  MoveC 664 to (45.79, 82.06, -1) mm, rotated rx -180 ry 0 rz 90 deg; joints [76.857, -17.355, 82.878, 0, 24.477, 76.857] to (20.03, 82.47, -1) mm, rotated rx -180 ry 0 rz 90 deg; joints [76.673, -17.853, 84.752, 0, 23.101, 76.673]
  MoveL 665 to (19.93, 74.92, -1) mm, rotated rx 180 ry 0 rz 90 deg; joints [76.425, -17.821, 84.63, 0, 23.192, 76.425]
  MoveL 666 to (19.93, 74.92, 2) mm, rotated rx 180 ry 0 rz 90 deg; joints [76.425, -17.975, 84.73, 0, 23.244, 76.425]
  Establecer velocidad (1000.0 mm/s)
  MoveL 667 to (19.93, 74.92, 10) mm, rotated rx 180 ry 0 rz 90 deg; joints [76.425, -18.384, 84.996, 0, 23.387, 76.425]
  Establecer velocidad (66.7 mm/s)
  MoveL 668 to (26.55, 73.47, 10) mm, rotated rx -180 ry 0 rz 90 deg; joints [76.43, -18.251, 84.495, 0, 23.756, 76.43]
  MoveL 669 to (26.55, 73.47, 2) mm, rotated rx 180 ry 0 rz 90 deg; joints [76.43, -17.843, 84.229, 0, 23.614, 76.43]
  MoveL 670 to (26.75, 74.97, 1.59) mm, rotated rx -180 ry 0 rz 90 deg; joints [76.48, -17.825, 84.227, 0, 23.598, 76.48]
  MoveL 671 to (26.59, 76.48, 1.19) mm, rotated rx -180 ry 0 rz 90 deg; joints [76.529, -17.815, 84.251, 0, 23.563, 76.529]
  MoveL 672 to (26.1, 77.92, 0.78) mm, rotated rx 180 ry 0 rz 90 deg; joints [76.572, -17.81, 84.298, 0, 23.512, 76.572]
  MoveL 673 to (25.3, 79.21, 0.38) mm, rotated rx 180 ry 0 rz 90 deg; joints [76.608, -17.81, 84.364, 0, 23.446, 76.608]
  MoveL 674 to (24.24, 80.3, -0.03) mm, rotated rx -180 ry 0 rz 90 deg; joints [76.635, -17.814, 84.446, 0, 23.369, 76.635]
  MoveL 675 to (22.96, 81.12, -0.44) mm, rotated rx 180 ry 0 rz 90 deg; joints [76.652, -17.821, 84.538, 0, 23.283, 76.652]
  MoveL 676 to (21.53, 81.64, -0.84) mm, rotated rx 180 ry 0 rz 90 deg; joints [76.658, -17.83, 84.636, 0, 23.194, 76.658]
  MoveL 677 to (20.02, 81.8, -1.25) mm, rotated rx 180 ry 0 rz 90 deg; joints [76.651, -17.838, 84.733, 0, 23.105, 76.651]
  MoveC 678 to (-5.39, 82.11, -1.25) mm, rotated rx 180 ry 0 rz 90 deg; joints [76.461, -18.297, 86.542, 0, 21.755, 76.461] to (-30.8, 82.31, -1.25) mm, rotated rx 180 ry 0 rz 90 deg; joints [76.261, -18.726, 88.313, 0, 20.412, 76.261]
  MoveC 679 to (-35.67, 81.83, -1.25) mm, rotated rx 180 ry 0 rz 90 deg; joints [76.205, -18.803, 88.641, 0, 20.162, 76.205] to (-40.33, 80.31, -1.25) mm, rotated rx -180 ry 0 rz 90 deg; joints [76.115, -18.871, 88.934, 0, 19.937, 76.115]
  MoveC 680 to (-44.55, 75.38, -1.25) mm, rotated rx 180 ry 0 rz 90 deg; joints [75.912, -18.918, 89.138, 0, 19.779, 75.912] to (-43.44, 68.99, -1.25) mm, rotated rx -180 ry 0 rz 90 deg; joints [75.705, -18.875, 88.953, 0, 19.922, 75.705]
  MoveC 681 to (-40.9, 66.02, -1.25) mm, rotated rx 180 ry 0 rz 90 deg; joints [75.627, -18.823, 88.727, 0, 20.096, 75.627] to (-37.82, 63.61, -1.25) mm, rotated rx 180 ry 0 rz 90 deg; joints [75.572, -18.763, 88.473, 0, 20.29, 75.572]
  MoveL 682 to (-14.69, 48.96, -1.25) mm, rotated rx 180 ry 0 rz 90 deg; joints [75.284, -18.314, 86.609, 0, 21.705, 75.284]
  MoveC 683 to (-10.76, 47.27, -1.25) mm, rotated rx -180 ry 0 rz 90 deg; joints [75.262, -18.238, 86.303, 0, 21.935, 75.262] to (-6.49, 46.9, -1.25) mm, rotated rx 180 ry 0 rz 90 deg; joints [75.287, -18.161, 85.996, 0, 22.165, 75.287]
  MoveL 684 to (63.97, 51.98, -1.25) mm, rotated rx 180 ry 0 rz 90 deg; joints [76.033, -16.822, 80.991, 0, 25.832, 76.033]
  MoveL 685 to (72.21, 52.56, -1.25) mm, rotated rx 180 ry 0 rz 90 deg; joints [76.117, -16.65, 80.385, 0, 26.266, 76.117]
  MoveC 686 to (77.75, 55.2, -1.25) mm, rotated rx 180 ry 0 rz 90 deg; joints [76.243, -16.545, 80.016, 0, 26.528, 76.243] to (80, 60.92, -1.25) mm, rotated rx -180 ry 0 rz 90 deg; joints [76.441, -16.526, 79.951, 0, 26.575, 76.441]
  MoveL 687 to (80, 72.47, -1.25) mm, rotated rx -180 ry 0 rz 90 deg; joints [76.806, -16.586, 80.159, 0, 26.426, 76.806]
  MoveC 688 to (77.62, 78.32, -1.25) mm, rotated rx -180 ry 0 rz 90 deg; joints [76.974, -16.667, 80.442, 0, 26.225, 76.974] to (71.82, 80.84, -1.25) mm, rotated rx -180 ry 0 rz 90 deg; joints [77.012, -16.803, 80.92, 0, 25.882, 77.012]
  MoveC 689 to (45.92, 81.38, -1.25) mm, rotated rx 180 ry 0 rz 90 deg; joints [76.836, -17.337, 82.848, 0, 24.488, 76.836] to (20.02, 81.8, -1.25) mm, rotated rx 180 ry 0 rz 90 deg; joints [76.651, -17.838, 84.733, 0, 23.105, 76.651]
  MoveL 690 to (19.92, 74.25, -1.25) mm, rotated rx 180 ry 0 rz 90 deg; joints [76.403, -17.806, 84.611, 0, 23.195, 76.403]
  MoveL 691 to (19.92, 74.25, 1.75) mm, rotated rx 180 ry 0 rz 90 deg; joints [76.403, -17.959, 84.711, 0, 23.248, 76.403]
  Establecer velocidad (1000.0 mm/s)
  MoveL 692 to (19.92, 74.25, 10) mm, rotated rx 180 ry 0 rz 90 deg; joints [76.403, -18.381, 84.985, 0, 23.395, 76.403]
  Establecer velocidad (66.7 mm/s)
  MoveL 693 to (38.36, 29.5, 10) mm, rotated rx -180 ry 0 rz 90 deg; joints [75.107, -17.799, 82.829, 0, 24.97, 75.107]
  MoveL 694 to (38.36, 29.5, 2) mm, rotated rx -180 ry 0 rz 90 deg; joints [75.107, -17.394, 82.562, 0, 24.831, 75.107]
  MoveL 695 to (38.51, 31.01, 1.59) mm, rotated rx -180 ry 0 rz 90 deg; joints [75.156, -17.378, 82.567, 0, 24.811, 75.156]
  MoveL 696 to (38.29, 32.51, 1.19) mm, rotated rx -180 ry 0 rz 90 deg; joints [75.203, -17.37, 82.599, 0, 24.771, 75.203]
  MoveL 697 to (37.74, 33.93, 0.78) mm, rotated rx 180 ry 0 rz 90 deg; joints [75.243, -17.368, 82.653, 0, 24.715, 75.243]
  MoveL 698 to (36.89, 35.19, 0.38) mm, rotated rx 180 ry 0 rz 90 deg; joints [75.277, -17.371, 82.725, 0, 24.646, 75.277]
  MoveL 699 to (35.78, 36.23, -0.03) mm, rotated rx -180 ry 0 rz 90 deg; joints [75.301, -17.378, 82.812, 0, 24.566, 75.301]
  MoveL 700 to (34.47, 37, -0.44) mm, rotated rx -180 ry 0 rz 90 deg; joints [75.314, -17.387, 82.909, 0, 24.478, 75.314]
  MoveL 701 to (33.02, 37.46, -0.84) mm, rotated rx 180 ry 0 rz 90 deg; joints [75.317, -17.397, 83.009, 0, 24.388, 75.317]
  MoveL 702 to (31.51, 37.56, -1.25) mm, rotated rx -180 ry 0 rz 90 deg; joints [75.307, -17.407, 83.107, 0, 24.3, 75.307]
  MoveL 703 to (7.58, 36.92, -1.25) mm, rotated rx 180 ry 0 rz 90 deg; joints [75.082, -17.859, 84.815, 0, 23.044, 75.082]
  MoveC 704 to (3.41, 36.01, -1.25) mm, rotated rx 180 ry 0 rz 90 deg; joints [75.016, -17.931, 85.093, 0, 22.838, 75.016] to (-0.13, 33.64, -1.25) mm, rotated rx -180 ry 0 rz 90 deg; joints [74.908, -17.984, 85.299, 0, 22.685, 74.908]
  MoveC 705 to (-2.38, 29.17, -1.25) mm, rotated rx -180 ry 0 rz 90 deg; joints [74.741, -18.003, 85.373, 0, 22.63, 74.741] to (-2.11, 24.17, -1.25) mm, rotated rx 180 ry 0 rz 90 deg; joints [74.581, -17.973, 85.256, 0, 22.717, 74.581]
  MoveL 706 to (-1.81, 23.22, -1.25) mm, rotated rx 180 ry 0 rz 90 deg; joints [74.552, -17.963, 85.217, 0, 22.746, 74.552]
  MoveL 707 to (3.68, 8.05, -1.25) mm, rotated rx 180 ry 0 rz 90 deg; joints [74.11, -17.784, 84.526, 0, 23.257, 74.11]
  MoveL 708 to (4.33, 6.33, -1.25) mm, rotated rx 180 ry 0 rz 90 deg; joints [74.06, -17.763, 84.446, 0, 23.317, 74.06]
  MoveC 709 to (5.69, 3.82, -1.25) mm, rotated rx -180 ry 0 rz 90 deg; joints [73.992, -17.724, 84.297, 0, 23.427, 73.992] to (7.69, 1.78, -1.25) mm, rotated rx -180 ry 0 rz 90 deg; joints [73.944, -17.675, 84.113, 0, 23.562, 73.944]
  MoveL 710 to (25.11, -11.75, -1.25) mm, rotated rx 180 ry 0 rz 90 deg; joints [73.673, -17.263, 82.579, 0, 24.685, 73.673]
  MoveC 711 to (32.35, -13.71, -1.25) mm, rotated rx -180 ry 0 rz 90 deg; joints [73.678, -17.107, 82.011, 0, 25.096, 73.678] to (38.84, -9.95, -1.25) mm, rotated rx 180 ry 0 rz 90 deg; joints [73.857, -16.998, 81.617, 0, 25.381, 73.857]
  MoveL 712 to (39.33, -9.33, -1.25) mm, rotated rx 180 ry 0 rz 90 deg; joints [73.881, -16.992, 81.594, 0, 25.397, 73.881]
  MoveL 713 to (62.07, 22.39, -1.25) mm, rotated rx 180 ry 0 rz 90 deg; joints [75.082, -16.701, 80.564, 0, 26.137, 75.082]
  MoveL 714 to (62.82, 23.49, -1.25) mm, rotated rx 180 ry 0 rz 90 deg; joints [75.123, -16.692, 80.53, 0, 26.162, 75.123]
  MoveC 715 to (64.55, 27.94, -1.25) mm, rotated rx 180 ry 0 rz 90 deg; joints [75.277, -16.68, 80.488, 0, 26.191, 75.277] to (64.19, 32.69, -1.25) mm, rotated rx 180 ry 0 rz 90 deg; joints [75.424, -16.714, 80.608, 0, 26.106, 75.424]
  MoveC 716 to (60.61, 36.69, -1.25) mm, rotated rx 180 ry 0 rz 90 deg; joints [75.521, -16.812, 80.952, 0, 25.859, 75.521] to (55.44, 38.13, -1.25) mm, rotated rx 180 ry 0 rz 90 deg; joints [75.525, -16.927, 81.364, 0, 25.564, 75.525]
  MoveL 717 to (53.54, 38.15, -1.25) mm, rotated rx -180 ry 0 rz 90 deg; joints [75.51, -16.967, 81.504, 0, 25.462, 75.51]
  MoveL 718 to (31.51, 37.56, -1.25) mm, rotated rx -180 ry 0 rz 90 deg; joints [75.307, -17.407, 83.107, 0, 24.3, 75.307]
  MoveL 719 to (31.71, 30.01, -1.25) mm, rotated rx -180 ry 0 rz 90 deg; joints [75.066, -17.364, 82.948, 0, 24.416, 75.066]
  MoveL 720 to (31.71, 30.01, 1.75) mm, rotated rx 180 ry 0 rz 90 deg; joints [75.066, -17.516, 83.048, 0, 24.468, 75.066]
  Establecer velocidad (1000.0 mm/s)
  MoveL 721 to (31.71, 30.01, 10) mm, rotated rx 180 ry 0 rz 90 deg; joints [75.066, -17.935, 83.323, 0, 24.612, 75.066]
  Establecer velocidad (66.7 mm/s)
  MoveL 722 to (72.21, -30.7, 10) mm, rotated rx 180 ry 0 rz 90 deg; joints [73.514, -16.719, 79.06, 0, 27.659, 73.514]
  MoveL 723 to (72.21, -30.7, 2) mm, rotated rx 180 ry 0 rz 90 deg; joints [73.514, -16.319, 78.791, 0, 27.527, 73.514]
  MoveL 724 to (73.71, -30.89, 1.59) mm, rotated rx 180 ry 0 rz 90 deg; joints [73.522, -16.263, 78.66, 0, 27.604, 73.522]
  MoveL 725 to (75.22, -30.71, 1.19) mm, rotated rx 180 ry 0 rz 90 deg; joints [73.541, -16.211, 78.536, 0, 27.675, 73.541]
  MoveL 726 to (76.65, -30.2, 0.78) mm, rotated rx 180 ry 0 rz 90 deg; joints [73.57, -16.161, 78.425, 0, 27.737, 73.57]
  MoveL 727 to (77.93, -29.38, 0.38) mm, rotated rx 180 ry 0 rz 90 deg; joints [73.607, -16.118, 78.332, 0, 27.786, 73.607]
  MoveL 728 to (79, -28.3, -0.03) mm, rotated rx -180 ry 0 rz 90 deg; joints [73.65, -16.08, 78.261, 0, 27.819, 73.65]
  MoveL 729 to (79.81, -27.01, -0.44) mm, rotated rx 180 ry 0 rz 90 deg; joints [73.697, -16.05, 78.215, 0, 27.836, 73.697]
  MoveL 730 to (80.31, -25.58, -0.84) mm, rotated rx 180 ry 0 rz 90 deg; joints [73.745, -16.028, 78.195, 0, 27.834, 73.745]
  MoveL 731 to (80.45, -24.06, -1.25) mm, rotated rx -180 ry 0 rz 90 deg; joints [73.793, -16.015, 78.204, 0, 27.811, 73.793]
  MoveL 732 to (80.45, -5.21, -1.25) mm, rotated rx 180 ry 0 rz 90 deg; joints [74.376, -16.136, 78.613, 0, 27.523, 74.376]
  MoveL 733 to (80.42, -3.53, -1.25) mm, rotated rx -180 ry 0 rz 90 deg; joints [74.427, -16.147, 78.651, 0, 27.496, 74.427]
  MoveC 734 to (80.02, -0.05, -1.25) mm, rotated rx 180 ry 0 rz 90 deg; joints [74.532, -16.178, 78.755, 0, 27.423, 74.532] to (78.95, 3.29, -1.25) mm, rotated rx 180 ry 0 rz 90 deg; joints [74.627, -16.222, 78.905, 0, 27.317, 74.627]
  MoveC 735 to (74.11, 7.51, -1.25) mm, rotated rx -180 ry 0 rz 90 deg; joints [74.717, -16.355, 79.359, 0, 26.995, 74.717] to (67.8, 6.36, -1.25) mm, rotated rx 180 ry 0 rz 90 deg; joints [74.627, -16.486, 79.811, 0, 26.675, 74.627]
  MoveC 736 to (65.35, 4.27, -1.25) mm, rotated rx 180 ry 0 rz 90 deg; joints [74.54, -16.526, 79.951, 0, 26.575, 74.54] to (63.25, 1.83, -1.25) mm, rotated rx -180 ry 0 rz 90 deg; joints [74.445, -16.557, 80.057, 0, 26.499, 74.445]
  MoveL 737 to (46.96, -20.52, -1.25) mm, rotated rx 180 ry 0 rz 90 deg; joints [73.599, -16.766, 80.793, 0, 25.974, 73.599]
  MoveC 738 to (45.17, -26.46, -1.25) mm, rotated rx 180 ry 0 rz 90 deg; joints [73.396, -16.767, 80.795, 0, 25.972, 73.396] to (47.5, -32.22, -1.25) mm, rotated rx -180 ry 0 rz 90 deg; joints [73.238, -16.682, 80.496, 0, 26.186, 73.238]
  MoveL 739 to (49.58, -34.59, -1.25) mm, rotated rx 180 ry 0 rz 90 deg; joints [73.183, -16.623, 80.288, 0, 26.334, 73.183]
  MoveL 740 to (62.07, -48.7, -1.25) mm, rotated rx 180 ry 0 rz 90 deg; joints [72.864, -16.26, 79.035, 0, 27.225, 72.864]
  MoveL 741 to (64.05, -50.95, -1.25) mm, rotated rx 180 ry 0 rz 90 deg; joints [72.814, -16.201, 78.834, 0, 27.367, 72.814]
  MoveC 742 to (66.41, -53.1, -1.25) mm, rotated rx -180 ry 0 rz 90 deg; joints [72.77, -16.134, 78.607, 0, 27.527, 72.77] to (69.17, -54.7, -1.25) mm, rotated rx -180 ry 0 rz 90 deg; joints [72.747, -16.061, 78.36, 0, 27.701, 72.747]
  MoveC 743 to (74.84, -54.84, -1.25) mm, rotated rx 180 ry 0 rz 90 deg; joints [72.797, -15.932, 77.928, 0, 28.005, 72.797] to (78.95, -50.94, -1.25) mm, rotated rx 180 ry 0 rz 90 deg; joints [72.955, -15.866, 77.706, 0, 28.16, 72.955]
  MoveC 744 to (79.99, -47.84, -1.25) mm, rotated rx 180 ry 0 rz 90 deg; joints [73.059, -15.864, 77.699, 0, 28.165, 73.059] to (80.41, -44.6, -1.25) mm, rotated rx 180 ry 0 rz 90 deg; joints [73.162, -15.877, 77.743, 0, 28.134, 73.162]
  MoveL 745 to (80.45, -43.12, -1.25) mm, rotated rx 180 ry 0 rz 90 deg; joints [73.208, -15.886, 77.773, 0, 28.113, 73.208]
  MoveL 746 to (80.45, -24.06, -1.25) mm, rotated rx -180 ry 0 rz 90 deg; joints [73.793, -16.015, 78.204, 0, 27.811, 73.793]
  MoveL 747 to (72.9, -24.06, -1.25) mm, rotated rx 180 ry 0 rz 90 deg; joints [73.725, -16.184, 78.777, 0, 27.407, 73.725]
  MoveL 748 to (72.9, -24.06, 1.75) mm, rotated rx -180 ry 0 rz 90 deg; joints [73.725, -16.334, 78.878, 0, 27.456, 73.725]
  Establecer velocidad (1000.0 mm/s)
  MoveL 749 to (72.9, -24.06, 10) mm, rotated rx 180 ry 0 rz 90 deg; joints [73.725, -16.747, 79.155, 0, 27.592, 73.725]
  Establecer velocidad (66.7 mm/s)
  MoveL 750 to (18.32, -73.74, 10) mm, rotated rx 180 ry 0 rz 90 deg; joints [71.653, -17.581, 82.045, 0, 25.536, 71.653]
  MoveL 751 to (18.32, -73.74, 2) mm, rotated rx 180 ry 0 rz 90 deg; joints [71.653, -17.177, 81.779, 0, 25.398, 71.653]
  MoveL 752 to (18.15, -75.25, 1.59) mm, rotated rx -180 ry 0 rz 90 deg; joints [71.604, -17.15, 81.741, 0, 25.409, 71.604]
  MoveL 753 to (18.35, -76.76, 1.19) mm, rotated rx -180 ry 0 rz 90 deg; joints [71.559, -17.115, 81.677, 0, 25.438, 71.559]
  MoveL 754 to (18.87, -78.18, 0.78) mm, rotated rx 180 ry 0 rz 90 deg; joints [71.52, -17.074, 81.591, 0, 25.484, 71.52]
  MoveL 755 to (19.7, -79.46, 0.38) mm, rotated rx 180 ry 0 rz 90 deg; joints [71.489, -17.028, 81.486, 0, 25.542, 71.489]
  MoveL 756 to (20.79, -80.51, -0.03) mm, rotated rx -180 ry 0 rz 90 deg; joints [71.467, -16.978, 81.368, 0, 25.611, 71.467]
  MoveL 757 to (22.09, -81.31, -0.44) mm, rotated rx -180 ry 0 rz 90 deg; joints [71.456, -16.926, 81.24, 0, 25.686, 71.456]
  MoveL 758 to (23.53, -81.79, -0.84) mm, rotated rx -180 ry 0 rz 90 deg; joints [71.456, -16.873, 81.11, 0, 25.762, 71.456]
  MoveL 759 to (25.04, -81.91, -1.25) mm, rotated rx 180 ry 0 rz 90 deg; joints [71.468, -16.82, 80.984, 0, 25.837, 71.468]
  MoveL 760 to (53.54, -81.62, -1.25) mm, rotated rx -180 ry 0 rz 90 deg; joints [71.769, -16.217, 78.888, 0, 27.329, 71.769]
  MoveL 761 to (55.06, -81.52, -1.25) mm, rotated rx 180 ry 0 rz 90 deg; joints [71.787, -16.184, 78.777, 0, 27.407, 71.787]
  MoveC 762 to (59.46, -80.25, -1.25) mm, rotated rx 180 ry 0 rz 90 deg; joints [71.87, -16.096, 78.478, 0, 27.618, 71.87] to (62.9, -77.23, -1.25) mm, rotated rx -180 ry 0 rz 90 deg; joints [71.997, -16.041, 78.294, 0, 27.748, 71.997]
  MoveC 763 to (63.97, -72.6, -1.25) mm, rotated rx 180 ry 0 rz 90 deg; joints [72.149, -16.051, 78.326, 0, 27.725, 72.149] to (62.62, -68.03, -1.25) mm, rotated rx -180 ry 0 rz 90 deg; joints [72.275, -16.114, 78.538, 0, 27.576, 72.275]
  MoveC 764 to (61.36, -66.14, -1.25) mm, rotated rx 180 ry 0 rz 90 deg; joints [72.321, -16.155, 78.678, 0, 27.477, 72.321] to (59.94, -64.36, -1.25) mm, rotated rx 180 ry 0 rz 90 deg; joints [72.362, -16.199, 78.827, 0, 27.372, 72.362]
  MoveL 765 to (32.58, -32.69, -1.25) mm, rotated rx 180 ry 0 rz 90 deg; joints [73.081, -16.988, 81.581, 0, 25.407, 73.081]
  MoveL 766 to (30.88, -30.8, -1.25) mm, rotated rx -180 ry 0 rz 90 deg; joints [73.125, -17.034, 81.747, 0, 25.287, 73.125]
  MoveL 767 to (30.8, -30.72, -1.25) mm, rotated rx 180 ry 0 rz 90 deg; joints [73.127, -17.036, 81.755, 0, 25.281, 73.127]
  MoveL 768 to (15.64, -18.58, -1.25) mm, rotated rx 180 ry 0 rz 90 deg; joints [73.367, -17.409, 83.117, 0, 24.293, 73.367]
  MoveL 769 to (14.69, -17.89, -1.25) mm, rotated rx -180 ry 0 rz 90 deg; joints [73.379, -17.432, 83.2, 0, 24.232, 73.379]
  MoveC 770 to (10.61, -16.09, -1.25) mm, rotated rx -180 ry 0 rz 90 deg; joints [73.398, -17.521, 83.53, 0, 23.99, 73.398] to (6.16, -16.06, -1.25) mm, rotated rx 180 ry 0 rz 90 deg; joints [73.356, -17.605, 83.849, 0, 23.757, 73.356]
  MoveC 771 to (1.83, -18.59, -1.25) mm, rotated rx 180 ry 0 rz 90 deg; joints [73.234, -17.673, 84.103, 0, 23.569, 73.234] to (-0.74, -22.9, -1.25) mm, rotated rx 180 ry 0 rz 90 deg; joints [73.07, -17.697, 84.193, 0, 23.503, 73.07]
  MoveL 772 to (-1.12, -24.17, -1.25) mm, rotated rx -180 ry 0 rz 90 deg; joints [73.026, -17.696, 84.192, 0, 23.504, 73.026]
  MoveL 773 to (-12.95, -68.7, -1.25) mm, rotated rx 180 ry 0 rz 90 deg; joints [71.483, -17.651, 84.021, 0, 23.63, 71.483]
  MoveL 774 to (-13.18, -69.65, -1.25) mm, rotated rx 180 ry 0 rz 90 deg; joints [71.45, -17.649, 84.015, 0, 23.635, 71.45]
  MoveC 775 to (-11.86, -77.67, -1.25) mm, rotated rx 180 ry 0 rz 90 deg; joints [71.21, -17.574, 83.731, 0, 23.843, 71.21] to (-4.97, -81.97, -1.25) mm, rotated rx -180 ry 0 rz 90 deg; joints [71.149, -17.416, 83.14, 0, 24.276, 71.149]
  MoveC 776 to (-3.18, -82.14, -1.25) mm, rotated rx 180 ry 0 rz 90 deg; joints [71.163, -17.38, 83.008, 0, 24.372, 71.163] to (-1.37, -82.19, -1.25) mm, rotated rx 180 ry 0 rz 90 deg; joints [71.181, -17.345, 82.879, 0, 24.466, 71.181]
  MoveL 777 to (25.04, -81.91, -1.25) mm, rotated rx 180 ry 0 rz 90 deg; joints [71.468, -16.82, 80.984, 0, 25.837, 71.468]
  MoveL 778 to (24.96, -74.36, -1.25) mm, rotated rx 180 ry 0 rz 90 deg; joints [71.702, -16.874, 81.172, 0, 25.701, 71.702]
  MoveL 779 to (24.96, -74.36, 1.75) mm, rotated rx -180 ry 0 rz 90 deg; joints [71.702, -17.025, 81.273, 0, 25.752, 71.702]
  Establecer velocidad (1000.0 mm/s)
  MoveL 780 to (24.96, -74.36, 10) mm, rotated rx -180 ry 0 rz 90 deg; joints [71.702, -17.441, 81.549, 0, 25.892, 71.702]
  Establecer velocidad (66.7 mm/s)
  MoveL 781 to (-60.08, -73.94, 10) mm, rotated rx -180 ry 0 rz 90 deg; joints [70.798, -19.029, 87.529, 0, 21.5, 70.798]
  MoveL 782 to (-60.08, -73.94, 2) mm, rotated rx 180 ry 0 rz 90 deg; joints [70.798, -18.616, 87.263, 0, 21.353, 70.798]
  MoveL 783 to (-60.25, -75.45, 1.59) mm, rotated rx -180 ry 0 rz 90 deg; joints [70.747, -18.589, 87.226, 0, 21.363, 70.747]
  MoveL 784 to (-60.06, -76.96, 1.19) mm, rotated rx 180 ry 0 rz 90 deg; joints [70.7, -18.556, 87.163, 0, 21.393, 70.7]
  MoveL 785 to (-59.53, -78.38, 0.78) mm, rotated rx 180 ry 0 rz 90 deg; joints [70.66, -18.518, 87.08, 0, 21.438, 70.66]
  MoveL 786 to (-58.7, -79.66, 0.38) mm, rotated rx -180 ry 0 rz 90 deg; joints [70.628, -18.476, 86.98, 0, 21.496, 70.628]
  MoveL 787 to (-57.62, -80.72, -0.03) mm, rotated rx -180 ry 0 rz 90 deg; joints [70.606, -18.43, 86.867, 0, 21.563, 70.606]
  MoveL 788 to (-56.32, -81.51, -0.44) mm, rotated rx -180 ry 0 rz 90 deg; joints [70.596, -18.383, 86.746, 0, 21.637, 70.596]
  MoveL 789 to (-54.88, -82, -0.84) mm, rotated rx 180 ry 0 rz 90 deg; joints [70.596, -18.335, 86.623, 0, 21.712, 70.596]
  MoveL 790 to (-53.37, -82.13, -1.25) mm, rotated rx 180 ry 0 rz 90 deg; joints [70.609, -18.288, 86.503, 0, 21.784, 70.609]
  MoveL 791 to (-36.48, -81.98, -1.25) mm, rotated rx 180 ry 0 rz 90 deg; joints [70.804, -17.996, 85.347, 0, 22.649, 70.804]
  MoveL 792 to (-35.19, -81.96, -1.25) mm, rotated rx -180 ry 0 rz 90 deg; joints [70.819, -17.973, 85.258, 0, 22.715, 70.819]
  MoveC 793 to (-28.29, -79.52, -1.25) mm, rotated rx 180 ry 0 rz 90 deg; joints [70.973, -17.865, 84.838, 0, 23.027, 70.973] to (-24.28, -73.41, -1.25) mm, rotated rx -180 ry 0 rz 90 deg; joints [71.212, -17.83, 84.705, 0, 23.126, 71.212]
  MoveL 794 to (-11.95, -26.06, -1.25) mm, rotated rx 180 ry 0 rz 90 deg; joints [72.858, -17.885, 84.916, 0, 22.969, 72.858]
  MoveL 795 to (-11.48, -24.17, -1.25) mm, rotated rx 180 ry 0 rz 90 deg; joints [72.924, -17.887, 84.924, 0, 22.963, 72.924]
  MoveC 796 to (-11.52, -18.64, -1.25) mm, rotated rx 180 ry 0 rz 90 deg; joints [73.102, -17.919, 85.045, 0, 22.873, 73.102] to (-14.07, -13.74, -1.25) mm, rotated rx 180 ry 0 rz 90 deg; joints [73.236, -17.991, 85.329, 0, 22.663, 73.236]
  MoveC 797 to (-18.74, -10.95, -1.25) mm, rotated rx 180 ry 0 rz 90 deg; joints [73.281, -18.09, 85.714, 0, 22.376, 73.281] to (-24.17, -10.71, -1.25) mm, rotated rx 180 ry 0 rz 90 deg; joints [73.235, -18.186, 86.097, 0, 22.089, 73.235]
  MoveL 798 to (-73.89, -21.27, -1.25) mm, rotated rx 180 ry 0 rz 90 deg; joints [72.38, -18.947, 89.266, 0, 19.681, 72.38]
  MoveC 799 to (-80.35, -25.23, -1.25) mm, rotated rx -180 ry 0 rz 90 deg; joints [72.179, -19.026, 89.613, 0, 19.413, 72.179] to (-82.88, -32.37, -1.25) mm, rotated rx 180 ry 0 rz 90 deg; joints [71.913, -19.029, 89.628, 0, 19.401, 71.913]
  MoveL 800 to (-82.89, -70.6, -1.25) mm, rotated rx -180 ry 0 rz 90 deg; joints [70.647, -18.832, 88.766, 0, 20.066, 70.647]
  MoveL 801 to (-82.86, -71.55, -1.25) mm, rotated rx 180 ry 0 rz 90 deg; joints [70.616, -18.826, 88.742, 0, 20.084, 70.616]
  MoveC 802 to (-79.34, -79.16, -1.25) mm, rotated rx 180 ry 0 rz 90 deg; joints [70.407, -18.729, 88.327, 0, 20.402, 70.407] to (-71.55, -82.27, -1.25) mm, rotated rx 180 ry 0 rz 90 deg; joints [70.396, -18.587, 87.731, 0, 20.857, 70.396]
  MoveL 803 to (-70.6, -82.27, -1.25) mm, rotated rx 180 ry 0 rz 90 deg; joints [70.407, -18.572, 87.667, 0, 20.905, 70.407]
  MoveL 804 to (-53.37, -82.13, -1.25) mm, rotated rx 180 ry 0 rz 90 deg; joints [70.609, -18.288, 86.503, 0, 21.784, 70.609]
  MoveL 805 to (-53.43, -74.57, -1.25) mm, rotated rx -180 ry 0 rz 90 deg; joints [70.852, -18.333, 86.688, 0, 21.646, 70.852]
  MoveL 806 to (-53.43, -74.57, 1.75) mm, rotated rx -180 ry 0 rz 90 deg; joints [70.852, -18.488, 86.788, 0, 21.7, 70.852]
  Establecer velocidad (1000.0 mm/s)
  MoveL 807 to (-53.43, -74.57, 10) mm, rotated rx -180 ry 0 rz 90 deg; joints [70.852, -18.913, 87.062, 0, 21.851, 70.852]
  Establecer velocidad (66.7 mm/s)
  MoveL 808 to (-74.65, 36.69, 10) mm, rotated rx 180 ry 0 rz 90 deg; joints [74.325, -19.808, 90.85, 0, 18.958, 74.325]
  MoveL 809 to (-74.65, 36.69, 2) mm, rotated rx 180 ry 0 rz 90 deg; joints [74.325, -19.389, 90.585, 0, 18.804, 74.325]
  MoveL 810 to (-76.15, 36.87, 1.59) mm, rotated rx -180 ry 0 rz 90 deg; joints [74.317, -19.39, 90.675, 0, 18.715, 74.317]
  MoveL 811 to (-77.66, 36.69, 1.19) mm, rotated rx 180 ry 0 rz 90 deg; joints [74.297, -19.39, 90.759, 0, 18.632, 74.297]
  MoveL 812 to (-79.09, 36.18, 0.78) mm, rotated rx -180 ry 0 rz 90 deg; joints [74.265, -19.387, 90.831, 0, 18.557, 74.265]
  MoveL 813 to (-80.37, 35.36, 0.38) mm, rotated rx 180 ry 0 rz 90 deg; joints [74.225, -19.381, 90.887, 0, 18.494, 74.225]
  MoveL 814 to (-81.44, 34.28, -0.03) mm, rotated rx 180 ry 0 rz 90 deg; joints [74.178, -19.371, 90.924, 0, 18.447, 74.178]
  MoveL 815 to (-82.25, 32.99, -0.44) mm, rotated rx 180 ry 0 rz 90 deg; joints [74.126, -19.356, 90.94, 0, 18.416, 74.126]
  MoveL 816 to (-82.75, 31.56, -0.84) mm, rotated rx 180 ry 0 rz 90 deg; joints [74.072, -19.336, 90.932, 0, 18.404, 74.072]
  MoveL 817 to (-82.89, 30.05, -1.25) mm, rotated rx 180 ry 0 rz 90 deg; joints [74.019, -19.31, 90.899, 0, 18.411, 74.019]
  MoveL 818 to (-82.89, 0.47, -1.25) mm, rotated rx 180 ry 0 rz 90 deg; joints [73.015, -19.183, 90.318, 0, 18.866, 73.015]
  MoveC 819 to (-78.88, -8.17, -1.25) mm, rotated rx -180 ry 0 rz 90 deg; joints [72.766, -19.085, 89.874, 0, 19.211, 72.766] to (-69.65, -10.55, -1.25) mm, rotated rx -180 ry 0 rz 90 deg; joints [72.782, -18.934, 89.208, 0, 19.726, 72.782]
  MoveL 820 to (-68.7, -10.38, -1.25) mm, rotated rx 180 ry 0 rz 90 deg; joints [72.797, -18.92, 89.148, 0, 19.772, 72.797]
  MoveL 821 to (-18.81, 1.12, -1.25) mm, rotated rx 180 ry 0 rz 90 deg; joints [73.673, -18.154, 85.969, 0, 22.185, 73.673]
  MoveC 822 to (-11.85, 6.18, -1.25) mm, rotated rx 180 ry 0 rz 90 deg; joints [73.904, -18.057, 85.585, 0, 22.472, 73.904] to (-10.67, 14.7, -1.25) mm, rotated rx -180 ry 0 rz 90 deg; joints [74.193, -18.079, 85.673, 0, 22.406, 74.193]
  MoveL 823 to (-10.92, 15.64, -1.25) mm, rotated rx 180 ry 0 rz 90 deg; joints [74.222, -18.088, 85.709, 0, 22.379, 74.222]
  MoveL 824 to (-17.82, 34.95, -1.25) mm, rotated rx 180 ry 0 rz 90 deg; joints [74.793, -18.303, 86.566, 0, 21.737, 74.793]
  MoveC 825 to (-19.66, 38.26, -1.25) mm, rotated rx 180 ry 0 rz 90 deg; joints [74.886, -18.35, 86.757, 0, 21.593, 74.886] to (-22.47, 40.8, -1.25) mm, rotated rx -180 ry 0 rz 90 deg; joints [74.945, -18.41, 87, 0, 21.41, 74.945]
  MoveL 826 to (-64.91, 68.04, -1.25) mm, rotated rx 180 ry 0 rz 90 deg; joints [75.485, -19.199, 90.39, 0, 18.809, 75.485]
  MoveL 827 to (-65.86, 68.57, -1.25) mm, rotated rx 180 ry 0 rz 90 deg; joints [75.495, -19.215, 90.463, 0, 18.752, 75.495]
  MoveL 828 to (-67, 69.12, -1.25) mm, rotated rx 180 ry 0 rz 90 deg; joints [75.504, -19.234, 90.549, 0, 18.685, 75.504]
  MoveC 829 to (-72.12, 70.31, -1.25) mm, rotated rx -180 ry 0 rz 90 deg; joints [75.499, -19.313, 90.912, 0, 18.401, 75.499] to (-77.23, 69.14, -1.25) mm, rotated rx -180 ry 0 rz 90 deg; joints [75.413, -19.382, 91.233, 0, 18.149, 75.413]
  MoveC 830 to (-81.3, 65.12, -1.25) mm, rotated rx -180 ry 0 rz 90 deg; joints [75.238, -19.425, 91.434, 0, 17.991, 75.238] to (-82.86, 59.62, -1.25) mm, rotated rx -180 ry 0 rz 90 deg; joints [75.034, -19.426, 91.44, 0, 17.986, 75.034]
  MoveL 831 to (-82.89, 58.28, -1.25) mm, rotated rx -180 ry 0 rz 90 deg; joints [74.987, -19.421, 91.418, 0, 18.003, 74.987]
  MoveL 832 to (-82.89, 30.05, -1.25) mm, rotated rx 180 ry 0 rz 90 deg; joints [74.019, -19.31, 90.899, 0, 18.411, 74.019]
  MoveL 833 to (-75.34, 30.05, -1.25) mm, rotated rx 180 ry 0 rz 90 deg; joints [74.093, -19.201, 90.396, 0, 18.804, 74.093]
  MoveL 834 to (-75.34, 30.05, 1.75) mm, rotated rx 180 ry 0 rz 90 deg; joints [74.093, -19.358, 90.497, 0, 18.861, 74.093]
  Establecer velocidad (1000.0 mm/s)
  MoveL 835 to (-75.34, 30.05, 10) mm, rotated rx -180 ry 0 rz 90 deg; joints [74.093, -19.791, 90.771, 0, 19.019, 74.093]
  Establecer velocidad (66.7 mm/s)
  MoveL 836 to (-74.06, 36.69, 10) mm, rotated rx -180 ry 0 rz 90 deg; joints [74.331, -19.799, 90.811, 0, 18.988, 74.331]
  MoveL 837 to (-74.06, 36.69, 1.75) mm, rotated rx 180 ry 0 rz 90 deg; joints [74.331, -19.367, 90.537, 0, 18.83, 74.331]
  MoveL 838 to (-75.56, 36.87, 1.34) mm, rotated rx -180 ry 0 rz 90 deg; joints [74.323, -19.368, 90.627, 0, 18.741, 74.323]
  MoveL 839 to (-77.07, 36.69, 0.94) mm, rotated rx 180 ry 0 rz 90 deg; joints [74.302, -19.368, 90.711, 0, 18.657, 74.302]
  MoveL 840 to (-78.5, 36.18, 0.53) mm, rotated rx -180 ry 0 rz 90 deg; joints [74.271, -19.366, 90.783, 0, 18.583, 74.271]
  MoveL 841 to (-79.78, 35.36, 0.12) mm, rotated rx 180 ry 0 rz 90 deg; joints [74.231, -19.36, 90.839, 0, 18.52, 74.231]
  MoveL 842 to (-80.85, 34.28, -0.28) mm, rotated rx 180 ry 0 rz 90 deg; joints [74.184, -19.349, 90.876, 0, 18.473, 74.184]
  MoveL 843 to (-81.66, 32.99, -0.69) mm, rotated rx 180 ry 0 rz 90 deg; joints [74.132, -19.334, 90.892, 0, 18.442, 74.132]
  MoveL 844 to (-82.16, 31.56, -1.09) mm, rotated rx -180 ry 0 rz 90 deg; joints [74.078, -19.314, 90.884, 0, 18.43, 74.078]
  MoveL 845 to (-82.3, 30.05, -1.5) mm, rotated rx -180 ry 0 rz 90 deg; joints [74.025, -19.289, 90.851, 0, 18.437, 74.025]
  MoveL 846 to (-82.3, 0.47, -1.5) mm, rotated rx 180 ry 0 rz 90 deg; joints [73.021, -19.161, 90.27, 0, 18.891, 73.021]
  MoveC 847 to (-78.45, -7.73, -1.5) mm, rotated rx 180 ry 0 rz 90 deg; joints [72.785, -19.067, 89.846, 0, 19.221, 72.785] to (-69.65, -9.93, -1.5) mm, rotated rx -180 ry 0 rz 90 deg; joints [72.803, -18.923, 89.212, 0, 19.711, 72.803]
  MoveL 848 to (-68.7, -9.76, -1.5) mm, rotated rx -180 ry 0 rz 90 deg; joints [72.818, -18.91, 89.152, 0, 19.758, 72.818]
  MoveL 849 to (-19.01, 1.69, -1.5) mm, rotated rx 180 ry 0 rz 90 deg; joints [73.69, -18.148, 85.986, 0, 22.162, 73.69]
  MoveC 850 to (-12.15, 6.89, -1.5) mm, rotated rx 180 ry 0 rz 90 deg; joints [73.925, -18.053, 85.612, 0, 22.441, 73.925] to (-11.48, 15.46, -1.5) mm, rotated rx -180 ry 0 rz 90 deg; joints [74.211, -18.084, 85.736, 0, 22.348, 74.211]
  MoveL 851 to (-18.37, 34.73, -1.5) mm, rotated rx -180 ry 0 rz 90 deg; joints [74.781, -18.299, 86.592, 0, 21.707, 74.781]
  MoveC 852 to (-20.09, 37.85, -1.5) mm, rotated rx 180 ry 0 rz 90 deg; joints [74.869, -18.343, 86.771, 0, 21.572, 74.869] to (-22.72, 40.24, -1.5) mm, rotated rx -180 ry 0 rz 90 deg; joints [74.924, -18.399, 86.998, 0, 21.401, 74.924]
  MoveL 853 to (-25.11, 41.81, -1.5) mm, rotated rx -180 ry 0 rz 90 deg; joints [74.955, -18.447, 87.194, 0, 21.253, 74.955]
  MoveL 854 to (-65.23, 67.54, -1.5) mm, rotated rx -180 ry 0 rz 90 deg; joints [75.465, -19.189, 90.394, 0, 18.795, 75.465]
  MoveC 855 to (-68.76, 69.14, -1.5) mm, rotated rx -180 ry 0 rz 90 deg; joints [75.489, -19.247, 90.659, 0, 18.588, 75.489] to (-72.61, 69.68, -1.5) mm, rotated rx 180 ry 0 rz 90 deg; joints [75.473, -19.305, 90.926, 0, 18.379, 75.473]
  MoveC 856 to (-78.16, 67.86, -1.5) mm, rotated rx 180 ry 0 rz 90 deg; joints [75.36, -19.377, 91.264, 0, 18.113, 75.36] to (-81.58, 63.11, -1.5) mm, rotated rx -180 ry 0 rz 90 deg; joints [75.166, -19.408, 91.409, 0, 17.999, 75.166]
  MoveC 857 to (-82.12, 60.85, -1.5) mm, rotated rx -180 ry 0 rz 90 deg; joints [75.083, -19.407, 91.404, 0, 18.003, 75.083] to (-82.3, 58.54, -1.5) mm, rotated rx 180 ry 0 rz 90 deg; joints [75.002, -19.401, 91.375, 0, 18.025, 75.002]
  MoveL 858 to (-82.3, 30.05, -1.5) mm, rotated rx -180 ry 0 rz 90 deg; joints [74.025, -19.289, 90.851, 0, 18.437, 74.025]
  MoveL 859 to (-74.75, 30.05, -1.5) mm, rotated rx 180 ry 0 rz 90 deg; joints [74.099, -19.179, 90.349, 0, 18.83, 74.099]
  MoveL 860 to (-74.75, 30.05, 1.5) mm, rotated rx 180 ry 0 rz 90 deg; joints [74.099, -19.336, 90.449, 0, 18.887, 74.099]
  Establecer velocidad (1000.0 mm/s)
  MoveL 861 to (-74.75, 30.05, 10) mm, rotated rx 180 ry 0 rz 90 deg; joints [74.099, -19.782, 90.732, 0, 19.05, 74.099]
  Establecer velocidad (66.7 mm/s)
  MoveL 862 to (-74.06, -45.34, 10) mm, rotated rx -180 ry 0 rz 90 deg; joints [71.579, -19.414, 89.127, 0, 20.287, 71.579]
  MoveL 863 to (-74.06, -45.34, 1.75) mm, rotated rx -180 ry 0 rz 90 deg; joints [71.579, -18.985, 88.854, 0, 20.131, 71.579]
  MoveL 864 to (-75.56, -45.16, 1.34) mm, rotated rx -180 ry 0 rz 90 deg; joints [71.568, -18.988, 88.945, 0, 20.043, 71.568]
  MoveL 865 to (-77.07, -45.34, 0.94) mm, rotated rx 180 ry 0 rz 90 deg; joints [71.546, -18.989, 89.028, 0, 19.961, 71.546]
  MoveL 866 to (-78.5, -45.85, 0.53) mm, rotated rx -180 ry 0 rz 90 deg; joints [71.513, -18.988, 89.099, 0, 19.889, 71.513]
  MoveL 867 to (-79.78, -46.67, 0.12) mm, rotated rx 180 ry 0 rz 90 deg; joints [71.472, -18.982, 89.152, 0, 19.83, 71.472]
  MoveL 868 to (-80.85, -47.74, -0.28) mm, rotated rx 180 ry 0 rz 90 deg; joints [71.424, -18.972, 89.186, 0, 19.786, 71.424]
  MoveL 869 to (-81.66, -49.03, -0.69) mm, rotated rx 180 ry 0 rz 90 deg; joints [71.372, -18.956, 89.197, 0, 19.759, 71.372]
  MoveL 870 to (-82.16, -50.47, -1.09) mm, rotated rx 180 ry 0 rz 90 deg; joints [71.319, -18.935, 89.184, 0, 19.751, 71.319]
  MoveL 871 to (-82.3, -51.98, -1.5) mm, rotated rx 180 ry 0 rz 90 deg; joints [71.267, -18.908, 89.146, 0, 19.762, 71.267]
  MoveL 872 to (-82.3, -70.6, -1.5) mm, rotated rx 180 ry 0 rz 90 deg; joints [70.653, -18.809, 88.718, 0, 20.091, 70.653]
  MoveL 873 to (-82.27, -71.55, -1.5) mm, rotated rx -180 ry 0 rz 90 deg; joints [70.623, -18.804, 88.694, 0, 20.11, 70.623]
  MoveC 874 to (-78.92, -78.74, -1.5) mm, rotated rx 180 ry 0 rz 90 deg; joints [70.426, -18.712, 88.301, 0, 20.411, 70.426] to (-71.55, -81.67, -1.5) mm, rotated rx 180 ry 0 rz 90 deg; joints [70.416, -18.578, 87.737, 0, 20.841, 70.416]
  MoveL 875 to (-70.6, -81.67, -1.5) mm, rotated rx 180 ry 0 rz 90 deg; joints [70.426, -18.562, 87.673, 0, 20.89, 70.426]
  MoveL 876 to (-36.48, -81.39, -1.5) mm, rotated rx -180 ry 0 rz 90 deg; joints [70.822, -17.987, 85.353, 0, 22.634, 70.822]
  MoveL 877 to (-35.23, -81.38, -1.5) mm, rotated rx 180 ry 0 rz 90 deg; joints [70.837, -17.965, 85.267, 0, 22.698, 70.837]
  MoveC 878 to (-28.67, -79.06, -1.5) mm, rotated rx 180 ry 0 rz 90 deg; joints [70.983, -17.862, 84.867, 0, 22.995, 70.983] to (-24.86, -73.24, -1.5) mm, rotated rx -180 ry 0 rz 90 deg; joints [71.211, -17.829, 84.74, 0, 23.089, 71.211]
  MoveL 879 to (-12.1, -24.17, -1.5) mm, rotated rx 180 ry 0 rz 90 deg; joints [72.918, -17.886, 84.959, 0, 22.927, 72.918]
  MoveC 880 to (-12.02, -19.21, -1.5) mm, rotated rx 180 ry 0 rz 90 deg; joints [73.079, -17.912, 85.06, 0, 22.852, 73.079] to (-14.03, -14.69, -1.5) mm, rotated rx 180 ry 0 rz 90 deg; joints [73.205, -17.973, 85.297, 0, 22.675, 73.205]
  MoveC 881 to (-18.63, -11.59, -1.5) mm, rotated rx -180 ry 0 rz 90 deg; joints [73.261, -18.071, 85.684, 0, 22.387, 73.261] to (-24.17, -11.31, -1.5) mm, rotated rx 180 ry 0 rz 90 deg; joints [73.216, -18.17, 86.076, 0, 22.094, 73.216]
  MoveL 882 to (-73.72, -21.83, -1.5) mm, rotated rx -180 ry 0 rz 90 deg; joints [72.363, -18.929, 89.235, 0, 19.694, 72.363]
  MoveC 883 to (-79.88, -25.6, -1.5) mm, rotated rx 180 ry 0 rz 90 deg; joints [72.171, -19.004, 89.566, 0, 19.438, 72.171] to (-82.29, -32.41, -1.5) mm, rotated rx 180 ry 0 rz 90 deg; joints [71.918, -19.007, 89.579, 0, 19.428, 71.918]
  MoveL 884 to (-82.3, -51.98, -1.5) mm, rotated rx 180 ry 0 rz 90 deg; joints [71.267, -18.908, 89.146, 0, 19.762, 71.267]
  MoveL 885 to (-74.75, -51.98, -1.5) mm, rotated rx -180 ry 0 rz 90 deg; joints [71.352, -18.792, 88.642, 0, 20.15, 71.352]
  MoveL 886 to (-74.75, -51.98, 1.5) mm, rotated rx 180 ry 0 rz 90 deg; joints [71.352, -18.948, 88.742, 0, 20.205, 71.352]
  Establecer velocidad (1000.0 mm/s)
  MoveL 887 to (-74.75, -51.98, 10) mm, rotated rx 180 ry 0 rz 90 deg; joints [71.352, -19.39, 89.025, 0, 20.365, 71.352]
  Establecer velocidad (66.7 mm/s)
  MoveL 888 to (18.2, -73.15, 10) mm, rotated rx 180 ry 0 rz 90 deg; joints [71.67, -17.587, 82.068, 0, 25.519, 71.67]
  MoveL 889 to (18.2, -73.15, 1.75) mm, rotated rx 180 ry 0 rz 90 deg; joints [71.67, -17.171, 81.793, 0, 25.377, 71.67]
  MoveL 890 to (18.03, -74.66, 1.34) mm, rotated rx 180 ry 0 rz 90 deg; joints [71.621, -17.143, 81.756, 0, 25.388, 71.621]
  MoveL 891 to (18.22, -76.17, 0.94) mm, rotated rx 180 ry 0 rz 90 deg; joints [71.576, -17.109, 81.692, 0, 25.417, 71.576]
  MoveL 892 to (18.75, -77.59, 0.53) mm, rotated rx 180 ry 0 rz 90 deg; joints [71.537, -17.068, 81.605, 0, 25.463, 71.537]
  MoveL 893 to (19.58, -78.87, 0.12) mm, rotated rx 180 ry 0 rz 90 deg; joints [71.506, -17.022, 81.501, 0, 25.521, 71.506]
  MoveL 894 to (20.67, -79.92, -0.28) mm, rotated rx 180 ry 0 rz 90 deg; joints [71.484, -16.972, 81.382, 0, 25.59, 71.484]
  MoveL 895 to (21.97, -80.72, -0.69) mm, rotated rx 180 ry 0 rz 90 deg; joints [71.473, -16.92, 81.255, 0, 25.665, 71.473]
  MoveL 896 to (23.41, -81.2, -1.09) mm, rotated rx 180 ry 0 rz 90 deg; joints [71.473, -16.867, 81.125, 0, 25.742, 71.473]
  MoveL 897 to (24.92, -81.32, -1.5) mm, rotated rx 180 ry 0 rz 90 deg; joints [71.485, -16.814, 80.998, 0, 25.816, 71.485]
  MoveL 898 to (46.91, -81.1, -1.5) mm, rotated rx -180 ry 0 rz 90 deg; joints [71.718, -16.352, 79.387, 0, 26.966, 71.718]
  MoveL 899 to (54.11, -81, -1.5) mm, rotated rx -180 ry 0 rz 90 deg; joints [71.794, -16.196, 78.853, 0, 27.344, 71.794]
  MoveC 900 to (57.84, -80.3, -1.5) mm, rotated rx -180 ry 0 rz 90 deg; joints [71.852, -16.119, 78.59, 0, 27.529, 71.852] to (61.12, -78.41, -1.5) mm, rotated rx -180 ry 0 rz 90 deg; joints [71.943, -16.06, 78.39, 0, 27.67, 71.943]
  MoveC 901 to (63.32, -74.34, -1.5) mm, rotated rx 180 ry 0 rz 90 deg; joints [72.089, -16.04, 78.324, 0, 27.716, 72.089] to (62.75, -69.74, -1.5) mm, rotated rx -180 ry 0 rz 90 deg; joints [72.224, -16.086, 78.478, 0, 27.608, 72.224]
  MoveC 902 to (61.37, -67.23, -1.5) mm, rotated rx -180 ry 0 rz 90 deg; joints [72.288, -16.134, 78.642, 0, 27.492, 72.288] to (59.65, -64.94, -1.5) mm, rotated rx 180 ry 0 rz 90 deg; joints [72.341, -16.189, 78.826, 0, 27.362, 72.341]
  MoveL 903 to (30.8, -31.59, -1.5) mm, rotated rx -180 ry 0 rz 90 deg; joints [73.099, -17.018, 81.727, 0, 25.291, 73.099]
  MoveL 904 to (29.97, -30.8, -1.5) mm, rotated rx 180 ry 0 rz 90 deg; joints [73.116, -17.04, 81.805, 0, 25.235, 73.116]
  MoveL 905 to (15.64, -19.32, -1.5) mm, rotated rx 180 ry 0 rz 90 deg; joints [73.343, -17.392, 83.092, 0, 24.3, 73.343]
  MoveL 906 to (14.48, -18.48, -1.5) mm, rotated rx -180 ry 0 rz 90 deg; joints [73.359, -17.42, 83.193, 0, 24.226, 73.359]
  MoveC 907 to (10.52, -16.68, -1.5) mm, rotated rx -180 ry 0 rz 90 deg; joints [73.378, -17.506, 83.516, 0, 23.99, 73.378] to (6.16, -16.68, -1.5) mm, rotated rx -180 ry 0 rz 90 deg; joints [73.337, -17.589, 83.827, 0, 23.762, 73.337]
  MoveC 908 to (2.13, -19.13, -1.5) mm, rotated rx 180 ry 0 rz 90 deg; joints [73.219, -17.651, 84.062, 0, 23.59, 73.219] to (-0.21, -23.22, -1.5) mm, rotated rx 180 ry 0 rz 90 deg; joints [73.065, -17.672, 84.14, 0, 23.532, 73.065]
  MoveL 909 to (-12.56, -69.65, -1.5) mm, rotated rx 180 ry 0 rz 90 deg; joints [71.457, -17.625, 83.963, 0, 23.662, 71.457]
  MoveC 910 to (-11.21, -77.54, -1.5) mm, rotated rx -180 ry 0 rz 90 deg; joints [71.222, -17.55, 83.68, 0, 23.87, 71.222] to (-4.26, -81.5, -1.5) mm, rotated rx -180 ry 0 rz 90 deg; joints [71.171, -17.393, 83.093, 0, 24.3, 71.171]
  MoveL 911 to (-3.32, -81.58, -1.5) mm, rotated rx 180 ry 0 rz 90 deg; joints [71.179, -17.374, 83.023, 0, 24.35, 71.179]
  MoveL 912 to (1.42, -81.57, -1.5) mm, rotated rx -180 ry 0 rz 90 deg; joints [71.23, -17.282, 82.686, 0, 24.596, 71.23]
  MoveL 913 to (24.92, -81.32, -1.5) mm, rotated rx 180 ry 0 rz 90 deg; joints [71.485, -16.814, 80.998, 0, 25.816, 71.485]
  MoveL 914 to (24.84, -73.77, -1.5) mm, rotated rx 180 ry 0 rz 90 deg; joints [71.719, -16.867, 81.187, 0, 25.681, 71.719]
  MoveL 915 to (24.84, -73.77, 1.5) mm, rotated rx 180 ry 0 rz 90 deg; joints [71.719, -17.019, 81.288, 0, 25.731, 71.719]
  Establecer velocidad (1000.0 mm/s)
  MoveL 916 to (24.84, -73.77, 10) mm, rotated rx -180 ry 0 rz 90 deg; joints [71.719, -17.447, 81.571, 0, 25.876, 71.719]
  Establecer velocidad (66.7 mm/s)
  MoveL 917 to (71.61, -30.65, 10) mm, rotated rx 180 ry 0 rz 90 deg; joints [73.51, -16.732, 79.106, 0, 27.626, 73.51]
  MoveL 918 to (71.61, -30.65, 1.75) mm, rotated rx 180 ry 0 rz 90 deg; joints [73.51, -16.32, 78.83, 0, 27.49, 73.51]
  MoveL 919 to (73.11, -30.83, 1.34) mm, rotated rx 180 ry 0 rz 90 deg; joints [73.518, -16.265, 78.698, 0, 27.567, 73.518]
  MoveL 920 to (74.62, -30.65, 0.94) mm, rotated rx -180 ry 0 rz 90 deg; joints [73.537, -16.212, 78.574, 0, 27.638, 73.537]
  MoveL 921 to (76.05, -30.14, 0.53) mm, rotated rx -180 ry 0 rz 90 deg; joints [73.566, -16.163, 78.463, 0, 27.7, 73.566]
  MoveL 922 to (77.34, -29.32, 0.12) mm, rotated rx -180 ry 0 rz 90 deg; joints [73.603, -16.119, 78.37, 0, 27.749, 73.603]
  MoveL 923 to (78.4, -28.24, -0.28) mm, rotated rx -180 ry 0 rz 90 deg; joints [73.646, -16.082, 78.299, 0, 27.782, 73.646]
  MoveL 924 to (79.21, -26.95, -0.69) mm, rotated rx 180 ry 0 rz 90 deg; joints [73.693, -16.052, 78.253, 0, 27.799, 73.693]
  MoveL 925 to (79.71, -25.52, -1.09) mm, rotated rx 180 ry 0 rz 90 deg; joints [73.742, -16.03, 78.233, 0, 27.796, 73.742]
  MoveL 926 to (79.85, -24.01, -1.5) mm, rotated rx -180 ry 0 rz 90 deg; joints [73.789, -16.016, 78.242, 0, 27.774, 73.789]
  MoveL 927 to (79.85, -4.36, -1.5) mm, rotated rx -180 ry 0 rz 90 deg; joints [74.397, -16.142, 78.668, 0, 27.474, 74.397]
  MoveC 928 to (79.58, -1.04, -1.5) mm, rotated rx -180 ry 0 rz 90 deg; joints [74.497, -16.169, 78.759, 0, 27.41, 74.497] to (78.77, 2.19, -1.5) mm, rotated rx 180 ry 0 rz 90 deg; joints [74.591, -16.207, 78.888, 0, 27.319, 74.591]
  MoveC 929 to (73.99, 6.76, -1.5) mm, rotated rx -180 ry 0 rz 90 deg; joints [74.692, -16.34, 79.344, 0, 26.996, 74.692] to (67.52, 5.44, -1.5) mm, rotated rx -180 ry 0 rz 90 deg; joints [74.595, -16.473, 79.804, 0, 26.669, 74.595]
  MoveL 930 to (67.24, 5.21, -1.5) mm, rotated rx -180 ry 0 rz 90 deg; joints [74.586, -16.478, 79.82, 0, 26.658, 74.586]
  MoveC 931 to (65.39, 3.49, -1.5) mm, rotated rx -180 ry 0 rz 90 deg; joints [74.516, -16.508, 79.924, 0, 26.584, 74.516] to (63.76, 1.54, -1.5) mm, rotated rx -180 ry 0 rz 90 deg; joints [74.441, -16.531, 80.005, 0, 26.526, 74.441]
  MoveL 932 to (47.49, -20.77, -1.5) mm, rotated rx -180 ry 0 rz 90 deg; joints [73.596, -16.741, 80.739, 0, 26.002, 73.596]
  MoveC 933 to (45.79, -26.4, -1.5) mm, rotated rx -180 ry 0 rz 90 deg; joints [73.404, -16.742, 80.742, 0, 26, 73.404] to (47.97, -31.87, -1.5) mm, rotated rx 180 ry 0 rz 90 deg; joints [73.253, -16.662, 80.46, 0, 26.202, 73.253]
  MoveL 934 to (48.68, -32.69, -1.5) mm, rotated rx 180 ry 0 rz 90 deg; joints [73.234, -16.641, 80.389, 0, 26.252, 73.234]
  MoveL 935 to (63.97, -49.97, -1.5) mm, rotated rx 180 ry 0 rz 90 deg; joints [72.843, -16.197, 78.855, 0, 27.342, 72.843]
  MoveL 936 to (65.04, -51.13, -1.5) mm, rotated rx -180 ry 0 rz 90 deg; joints [72.818, -16.165, 78.747, 0, 27.418, 72.818]
  MoveC 937 to (67.09, -52.88, -1.5) mm, rotated rx -180 ry 0 rz 90 deg; joints [72.783, -16.108, 78.552, 0, 27.556, 72.783] to (69.47, -54.16, -1.5) mm, rotated rx 180 ry 0 rz 90 deg; joints [72.767, -16.046, 78.342, 0, 27.704, 72.767]
  MoveC 938 to (74.98, -54.05, -1.5) mm, rotated rx -180 ry 0 rz 90 deg; joints [72.822, -15.922, 77.927, 0, 27.995, 72.822] to (78.73, -50.02, -1.5) mm, rotated rx -180 ry 0 rz 90 deg; joints [72.981, -15.865, 77.736, 0, 28.129, 72.981]
  MoveC 939 to (79.57, -46.88, -1.5) mm, rotated rx -180 ry 0 rz 90 deg; joints [73.085, -15.868, 77.745, 0, 28.123, 73.085] to (79.85, -43.65, -1.5) mm, rotated rx 180 ry 0 rz 90 deg; joints [73.186, -15.884, 77.798, 0, 28.085, 73.186]
  MoveL 940 to (79.85, -24.01, -1.5) mm, rotated rx -180 ry 0 rz 90 deg; joints [73.789, -16.016, 78.242, 0, 27.774, 73.789]
  MoveL 941 to (72.3, -24.01, -1.5) mm, rotated rx -180 ry 0 rz 90 deg; joints [73.722, -16.185, 78.815, 0, 27.37, 73.722]
  MoveL 942 to (72.3, -24.01, 1.5) mm, rotated rx -180 ry 0 rz 90 deg; joints [73.722, -16.336, 78.916, 0, 27.419, 73.722]
  Establecer velocidad (1000.0 mm/s)
  MoveL 943 to (72.3, -24.01, 10) mm, rotated rx 180 ry 0 rz 90 deg; joints [73.722, -16.761, 79.201, 0, 27.559, 73.722]
  Establecer velocidad (66.7 mm/s)
  MoveL 944 to (39.51, 6.06, 10) mm, rotated rx 180 ry 0 rz 90 deg; joints [74.37, -17.646, 82.277, 0, 25.369, 74.37]
  MoveL 945 to (39.51, 6.06, 1.75) mm, rotated rx -180 ry 0 rz 90 deg; joints [74.37, -17.229, 82.002, 0, 25.227, 74.37]
  MoveL 946 to (40.63, 5.03, 1.34) mm, rotated rx -180 ry 0 rz 90 deg; joints [74.347, -17.18, 81.886, 0, 25.294, 74.347]
  MoveL 947 to (41.96, 4.3, 0.94) mm, rotated rx 180 ry 0 rz 90 deg; joints [74.336, -17.128, 81.759, 0, 25.368, 74.336]
  MoveL 948 to (43.42, 3.88, 0.53) mm, rotated rx -180 ry 0 rz 90 deg; joints [74.336, -17.075, 81.63, 0, 25.445, 74.336]
  MoveL 949 to (44.94, 3.79, 0.12) mm, rotated rx -180 ry 0 rz 90 deg; joints [74.346, -17.023, 81.503, 0, 25.52, 74.346]
  MoveL 950 to (46.44, 4.05, -0.28) mm, rotated rx 180 ry 0 rz 90 deg; joints [74.368, -16.973, 81.384, 0, 25.589, 74.368]
  MoveL 951 to (47.84, 4.63, -0.69) mm, rotated rx 180 ry 0 rz 90 deg; joints [74.398, -16.927, 81.279, 0, 25.648, 74.398]
  MoveL 952 to (49.08, 5.5, -1.09) mm, rotated rx 180 ry 0 rz 90 deg; joints [74.437, -16.885, 81.192, 0, 25.694, 74.437]
  MoveL 953 to (50.08, 6.65, -1.5) mm, rotated rx -180 ry 0 rz 90 deg; joints [74.482, -16.851, 81.128, 0, 25.723, 74.482]
  MoveL 954 to (61.29, 22.27, -1.5) mm, rotated rx -180 ry 0 rz 90 deg; joints [75.071, -16.705, 80.611, 0, 26.093, 75.071]
  MoveL 955 to (61.93, 23.22, -1.5) mm, rotated rx -180 ry 0 rz 90 deg; joints [75.106, -16.697, 80.583, 0, 26.114, 75.106]
  MoveC 956 to (63.35, 25.93, -1.5) mm, rotated rx -180 ry 0 rz 90 deg; joints [75.204, -16.681, 80.53, 0, 26.152, 75.204] to (64.09, 28.9, -1.5) mm, rotated rx 180 ry 0 rz 90 deg; joints [75.304, -16.682, 80.533, 0, 26.149, 75.304]
  MoveC 957 to (63.15, 33.42, -1.5) mm, rotated rx 180 ry 0 rz 90 deg; joints [75.439, -16.727, 80.692, 0, 26.036, 75.439] to (59.7, 36.48, -1.5) mm, rotated rx 180 ry 0 rz 90 deg; joints [75.507, -16.817, 81.008, 0, 25.809, 75.507]
  MoveC 958 to (57.15, 37.3, -1.5) mm, rotated rx -180 ry 0 rz 90 deg; joints [75.513, -16.875, 81.212, 0, 25.662, 75.513] to (54.49, 37.56, -1.5) mm, rotated rx -180 ry 0 rz 90 deg; joints [75.499, -16.931, 81.414, 0, 25.517, 75.499]
  MoveL 959 to (53.54, 37.56, -1.5) mm, rotated rx -180 ry 0 rz 90 deg; joints [75.491, -16.951, 81.485, 0, 25.466, 75.491]
  MoveL 960 to (7.11, 36.27, -1.5) mm, rotated rx 180 ry 0 rz 90 deg; joints [75.057, -17.852, 84.827, 0, 23.024, 75.057]
  MoveC 961 to (3.1, 35.24, -1.5) mm, rotated rx 180 ry 0 rz 90 deg; joints [74.988, -17.92, 85.092, 0, 22.828, 74.988] to (-0.17, 32.69, -1.5) mm, rotated rx 180 ry 0 rz 90 deg; joints [74.876, -17.967, 85.275, 0, 22.692, 74.876]
  MoveC 962 to (-1.88, 28.59, -1.5) mm, rotated rx 180 ry 0 rz 90 deg; joints [74.727, -17.978, 85.318, 0, 22.66, 74.727] to (-1.48, 24.17, -1.5) mm, rotated rx -180 ry 0 rz 90 deg; joints [74.586, -17.949, 85.203, 0, 22.745, 74.586]
  MoveL 963 to (-1.17, 23.22, -1.5) mm, rotated rx -180 ry 0 rz 90 deg; joints [74.558, -17.938, 85.163, 0, 22.775, 74.558]
  MoveL 964 to (4.89, 6.55, -1.5) mm, rotated rx 180 ry 0 rz 90 deg; joints [74.072, -17.741, 84.402, 0, 23.339, 74.072]
  MoveC 965 to (6.12, 4.24, -1.5) mm, rotated rx -180 ry 0 rz 90 deg; joints [74.009, -17.705, 84.267, 0, 23.438, 74.009] to (7.94, 2.35, -1.5) mm, rotated rx -180 ry 0 rz 90 deg; joints [73.965, -17.661, 84.098, 0, 23.563, 73.965]
  MoveL 966 to (10.34, 0.47, -1.5) mm, rotated rx -180 ry 0 rz 90 deg; joints [73.927, -17.605, 83.889, 0, 23.717, 73.927]
  MoveL 967 to (25.4, -11.25, -1.5) mm, rotated rx 180 ry 0 rz 90 deg; joints [73.692, -17.248, 82.56, 0, 24.688, 73.692]
  MoveC 968 to (32.05, -13.14, -1.5) mm, rotated rx 180 ry 0 rz 90 deg; joints [73.694, -17.104, 82.037, 0, 25.068, 73.694] to (38.14, -9.86, -1.5) mm, rotated rx 180 ry 0 rz 90 deg; joints [73.854, -17, 81.662, 0, 25.338, 73.854]
  MoveL 969 to (38.85, -9, -1.5) mm, rotated rx 180 ry 0 rz 90 deg; joints [73.887, -16.991, 81.628, 0, 25.363, 73.887]
  MoveL 970 to (50.08, 6.65, -1.5) mm, rotated rx -180 ry 0 rz 90 deg; joints [74.482, -16.851, 81.128, 0, 25.723, 74.482]
  MoveL 971 to (43.94, 11.05, -1.5) mm, rotated rx -180 ry 0 rz 90 deg; joints [74.567, -17.002, 81.67, 0, 25.333, 74.567]
  MoveL 972 to (43.94, 11.05, 1.5) mm, rotated rx 180 ry 0 rz 90 deg; joints [74.567, -17.154, 81.771, 0, 25.383, 74.567]
  Establecer velocidad (1000.0 mm/s)
  MoveL 973 to (43.94, 11.05, 10) mm, rotated rx 180 ry 0 rz 90 deg; joints [74.567, -17.583, 82.054, 0, 25.529, 74.567]
  Establecer velocidad (66.7 mm/s)
  MoveL 974 to (26.9, 72.87, 10) mm, rotated rx 180 ry 0 rz 90 deg; joints [76.413, -18.241, 84.459, 0, 23.782, 76.413]
  MoveL 975 to (26.9, 72.87, 1.75) mm, rotated rx 180 ry 0 rz 90 deg; joints [76.413, -17.821, 84.185, 0, 23.636, 76.413]
  MoveL 976 to (27.11, 74.37, 1.34) mm, rotated rx -180 ry 0 rz 90 deg; joints [76.464, -17.803, 84.183, 0, 23.62, 76.464]
  MoveL 977 to (26.95, 75.89, 0.94) mm, rotated rx 180 ry 0 rz 90 deg; joints [76.512, -17.792, 84.207, 0, 23.585, 76.512]
  MoveL 978 to (26.45, 77.32, 0.53) mm, rotated rx 180 ry 0 rz 90 deg; joints [76.555, -17.788, 84.254, 0, 23.534, 76.555]
  MoveL 979 to (25.66, 78.62, 0.12) mm, rotated rx 180 ry 0 rz 90 deg; joints [76.591, -17.788, 84.32, 0, 23.468, 76.591]
  MoveL 980 to (24.59, 79.7, -0.28) mm, rotated rx -180 ry 0 rz 90 deg; joints [76.618, -17.792, 84.401, 0, 23.391, 76.618]
  MoveL 981 to (23.31, 80.52, -0.69) mm, rotated rx -180 ry 0 rz 90 deg; joints [76.635, -17.799, 84.494, 0, 23.305, 76.635]
  MoveL 982 to (21.88, 81.04, -1.09) mm, rotated rx 180 ry 0 rz 90 deg; joints [76.641, -17.807, 84.592, 0, 23.216, 76.641]
  MoveL 983 to (20.38, 81.2, -1.5) mm, rotated rx 180 ry 0 rz 90 deg; joints [76.634, -17.816, 84.689, 0, 23.127, 76.634]
  MoveC 984 to (-5.21, 81.51, -1.5) mm, rotated rx 180 ry 0 rz 90 deg; joints [76.442, -18.279, 86.511, 0, 21.768, 76.442] to (-30.8, 81.71, -1.5) mm, rotated rx 180 ry 0 rz 90 deg; joints [76.241, -18.71, 88.295, 0, 20.416, 76.241]
  MoveC 985 to (-35.37, 81.28, -1.5) mm, rotated rx 180 ry 0 rz 90 deg; joints [76.189, -18.782, 88.602, 0, 20.18, 76.189] to (-39.76, 79.94, -1.5) mm, rotated rx 180 ry 0 rz 90 deg; joints [76.107, -18.847, 88.881, 0, 19.967, 76.107]
  MoveC 986 to (-43.91, 75.24, -1.5) mm, rotated rx 180 ry 0 rz 90 deg; joints [75.912, -18.894, 89.084, 0, 19.81, 75.912] to (-42.79, 69.07, -1.5) mm, rotated rx 180 ry 0 rz 90 deg; joints [75.713, -18.852, 88.901, 0, 19.951, 75.713]
  MoveC 987 to (-40.64, 66.61, -1.5) mm, rotated rx 180 ry 0 rz 90 deg; joints [75.649, -18.808, 88.711, 0, 20.097, 75.649] to (-38.1, 64.56, -1.5) mm, rotated rx 180 ry 0 rz 90 deg; joints [75.601, -18.759, 88.501, 0, 20.258, 75.601]
  MoveL 988 to (-36.48, 63.47, -1.5) mm, rotated rx -180 ry 0 rz 90 deg; joints [75.579, -18.728, 88.371, 0, 20.357, 75.579]
  MoveL 989 to (-14.32, 49.44, -1.5) mm, rotated rx 180 ry 0 rz 90 deg; joints [75.303, -18.297, 86.584, 0, 21.713, 75.303]
  MoveC 990 to (-10.56, 47.83, -1.5) mm, rotated rx 180 ry 0 rz 90 deg; joints [75.282, -18.224, 86.291, 0, 21.933, 75.282] to (-6.49, 47.48, -1.5) mm, rotated rx 180 ry 0 rz 90 deg; joints [75.306, -18.151, 85.999, 0, 22.152, 75.306]
  MoveL 991 to (65.86, 52.72, -1.5) mm, rotated rx 180 ry 0 rz 90 deg; joints [76.072, -16.774, 80.855, 0, 25.919, 76.072]
  MoveL 992 to (72.14, 53.15, -1.5) mm, rotated rx 180 ry 0 rz 90 deg; joints [76.135, -16.642, 80.392, 0, 26.25, 76.135]
  MoveC 993 to (77.31, 55.61, -1.5) mm, rotated rx -180 ry 0 rz 90 deg; joints [76.253, -16.544, 80.049, 0, 26.495, 76.253] to (79.41, 60.93, -1.5) mm, rotated rx 180 ry 0 rz 90 deg; joints [76.437, -16.526, 79.988, 0, 26.538, 76.437]
  MoveL 994 to (79.41, 72.49, -1.5) mm, rotated rx -180 ry 0 rz 90 deg; joints [76.803, -16.586, 80.196, 0, 26.39, 76.803]
  MoveC 995 to (77.07, 78, -1.5) mm, rotated rx -180 ry 0 rz 90 deg; joints [76.96, -16.664, 80.468, 0, 26.196, 76.96] to (71.55, 80.28, -1.5) mm, rotated rx -180 ry 0 rz 90 deg; joints [76.992, -16.793, 80.923, 0, 25.87, 76.992]
  MoveC 996 to (45.96, 80.79, -1.5) mm, rotated rx 180 ry 0 rz 90 deg; joints [76.817, -17.321, 82.827, 0, 24.494, 76.817] to (20.38, 81.2, -1.5) mm, rotated rx 180 ry 0 rz 90 deg; joints [76.634, -17.816, 84.689, 0, 23.127, 76.634]
  MoveL 997 to (20.27, 73.65, -1.5) mm, rotated rx -180 ry 0 rz 90 deg; joints [76.386, -17.784, 84.567, 0, 23.217, 76.386]
  MoveL 998 to (20.27, 73.65, 1.5) mm, rotated rx 180 ry 0 rz 90 deg; joints [76.386, -17.937, 84.667, 0, 23.27, 76.386]
  Establecer velocidad (1000.0 mm/s)
  MoveL 999 to (20.27, 73.65, 10) mm, rotated rx 180 ry 0 rz 90 deg; joints [76.386, -18.371, 84.95, 0, 23.422, 76.386]
  Establecer velocidad (66.7 mm/s)
  MoveL 1000 to (26.89, 72.32, 10) mm, rotated rx 180 ry 0 rz 90 deg; joints [76.395, -18.239, 84.45, 0, 23.789, 76.395]
  MoveL 1001 to (26.89, 72.32, 1.5) mm, rotated rx 180 ry 0 rz 90 deg; joints [76.395, -17.806, 84.168, 0, 23.638, 76.395]
  MoveL 1002 to (27.1, 73.83, 1.09) mm, rotated rx -180 ry 0 rz 90 deg; joints [76.446, -17.788, 84.166, 0, 23.623, 76.446]
  MoveL 1003 to (26.94, 75.34, 0.69) mm, rotated rx 180 ry 0 rz 90 deg; joints [76.494, -17.777, 84.19, 0, 23.588, 76.494]
  MoveL 1004 to (26.44, 76.77, 0.28) mm, rotated rx -180 ry 0 rz 90 deg; joints [76.537, -17.773, 84.237, 0, 23.536, 76.537]
  MoveL 1005 to (25.65, 78.07, -0.12) mm, rotated rx -180 ry 0 rz 90 deg; joints [76.573, -17.773, 84.303, 0, 23.47, 76.573]
  MoveL 1006 to (24.58, 79.15, -0.53) mm, rotated rx -180 ry 0 rz 90 deg; joints [76.6, -17.777, 84.384, 0, 23.393, 76.6]
  MoveL 1007 to (23.3, 79.98, -0.94) mm, rotated rx -180 ry 0 rz 90 deg; joints [76.617, -17.784, 84.477, 0, 23.307, 76.617]
  MoveL 1008 to (21.88, 80.5, -1.34) mm, rotated rx -180 ry 0 rz 90 deg; joints [76.623, -17.792, 84.574, 0, 23.218, 76.623]
  MoveL 1009 to (20.37, 80.66, -1.75) mm, rotated rx 180 ry 0 rz 90 deg; joints [76.616, -17.801, 84.672, 0, 23.129, 76.616]
  MoveC 1010 to (-5.21, 80.97, -1.75) mm, rotated rx 180 ry 0 rz 90 deg; joints [76.424, -18.264, 86.494, 0, 21.77, 76.424] to (-30.8, 81.16, -1.75) mm, rotated rx -180 ry 0 rz 90 deg; joints [76.222, -18.695, 88.277, 0, 20.418, 76.222]
  MoveC 1011 to (-35.14, 80.77, -1.75) mm, rotated rx -180 ry 0 rz 90 deg; joints [76.173, -18.764, 88.569, 0, 20.194, 76.173] to (-39.33, 79.55, -1.75) mm, rotated rx -180 ry 0 rz 90 deg; joints [76.097, -18.826, 88.836, 0, 19.99, 76.097]
  MoveC 1012 to (-43.35, 74.8, -1.75) mm, rotated rx 180 ry 0 rz 90 deg; joints [75.902, -18.871, 89.03, 0, 19.841, 75.902] to (-41.88, 68.75, -1.75) mm, rotated rx 180 ry 0 rz 90 deg; joints [75.71, -18.823, 88.825, 0, 19.998, 75.71]
  MoveC 1013 to (-39.45, 66.31, -1.75) mm, rotated rx -180 ry 0 rz 90 deg; joints [75.649, -18.775, 88.616, 0, 20.159, 75.649] to (-36.68, 64.25, -1.75) mm, rotated rx 180 ry 0 rz 90 deg; joints [75.603, -18.722, 88.39, 0, 20.332, 75.603]
  MoveL 1014 to (-13.99, 49.88, -1.75) mm, rotated rx -180 ry 0 rz 90 deg; joints [75.32, -18.28, 86.56, 0, 21.72, 75.32]
  MoveC 1015 to (-10.41, 48.35, -1.75) mm, rotated rx 180 ry 0 rz 90 deg; joints [75.301, -18.211, 86.282, 0, 21.929, 75.301] to (-6.54, 48.02, -1.75) mm, rotated rx -180 ry 0 rz 90 deg; joints [75.323, -18.141, 86.004, 0, 22.137, 75.323]
  MoveL 1016 to (3.71, 48.8, -1.75) mm, rotated rx -180 ry 0 rz 90 deg; joints [75.437, -17.961, 85.294, 0, 22.667, 75.437]
  MoveL 1017 to (70.6, 53.58, -1.75) mm, rotated rx -180 ry 0 rz 90 deg; joints [76.136, -16.665, 80.508, 0, 26.157, 76.136]
  MoveL 1018 to (72.03, 53.67, -1.75) mm, rotated rx 180 ry 0 rz 90 deg; joints [76.15, -16.635, 80.402, 0, 26.233, 76.15]
  MoveC 1019 to (76.89, 55.94, -1.75) mm, rotated rx -180 ry 0 rz 90 deg; joints [76.26, -16.542, 80.079, 0, 26.464, 76.26] to (78.86, 60.93, -1.75) mm, rotated rx 180 ry 0 rz 90 deg; joints [76.433, -16.526, 80.021, 0, 26.505, 76.433]
  MoveL 1020 to (78.86, 72.49, -1.75) mm, rotated rx -180 ry 0 rz 90 deg; joints [76.798, -16.585, 80.229, 0, 26.357, 76.798]
  MoveC 1021 to (76.81, 77.52, -1.75) mm, rotated rx 180 ry 0 rz 90 deg; joints [76.943, -16.655, 80.472, 0, 26.183, 76.943] to (71.83, 79.68, -1.75) mm, rotated rx -180 ry 0 rz 90 deg; joints [76.975, -16.772, 80.883, 0, 25.888, 76.975]
  MoveC 1022 to (46.1, 80.23, -1.75) mm, rotated rx 180 ry 0 rz 90 deg; joints [76.8, -17.303, 82.799, 0, 24.504, 76.8] to (20.37, 80.66, -1.75) mm, rotated rx 180 ry 0 rz 90 deg; joints [76.616, -17.801, 84.672, 0, 23.129, 76.616]
  MoveL 1023 to (20.26, 73.11, -1.75) mm, rotated rx 180 ry 0 rz 90 deg; joints [76.368, -17.769, 84.549, 0, 23.219, 76.368]
  MoveL 1024 to (20.26, 73.11, 1.25) mm, rotated rx 180 ry 0 rz 90 deg; joints [76.368, -17.922, 84.65, 0, 23.272, 76.368]
  Establecer velocidad (1000.0 mm/s)
  MoveL 1025 to (20.26, 73.11, 10) mm, rotated rx 180 ry 0 rz 90 deg; joints [76.368, -18.369, 84.941, 0, 23.428, 76.368]
  Establecer velocidad (66.7 mm/s)
  MoveL 1026 to (37.66, 28.35, 10) mm, rotated rx 180 ry 0 rz 90 deg; joints [75.064, -17.807, 82.858, 0, 24.949, 75.064]
  MoveL 1027 to (37.66, 28.35, 1.5) mm, rotated rx 180 ry 0 rz 90 deg; joints [75.064, -17.377, 82.575, 0, 24.802, 75.064]
  MoveL 1028 to (37.8, 29.86, 1.09) mm, rotated rx 180 ry 0 rz 90 deg; joints [75.114, -17.361, 82.58, 0, 24.781, 75.114]
  MoveL 1029 to (37.58, 31.36, 0.69) mm, rotated rx 180 ry 0 rz 90 deg; joints [75.16, -17.353, 82.612, 0, 24.741, 75.16]
  MoveL 1030 to (37.03, 32.78, 0.28) mm, rotated rx -180 ry 0 rz 90 deg; joints [75.201, -17.351, 82.666, 0, 24.685, 75.201]
  MoveL 1031 to (36.18, 34.04, -0.12) mm, rotated rx -180 ry 0 rz 90 deg; joints [75.234, -17.354, 82.738, 0, 24.615, 75.234]
  MoveL 1032 to (35.07, 35.08, -0.53) mm, rotated rx -180 ry 0 rz 90 deg; joints [75.258, -17.36, 82.825, 0, 24.535, 75.258]
  MoveL 1033 to (33.76, 35.85, -0.94) mm, rotated rx 180 ry 0 rz 90 deg; joints [75.271, -17.37, 82.922, 0, 24.448, 75.271]
  MoveL 1034 to (32.31, 36.31, -1.34) mm, rotated rx 180 ry 0 rz 90 deg; joints [75.274, -17.38, 83.022, 0, 24.358, 75.274]
  MoveL 1035 to (30.8, 36.41, -1.75) mm, rotated rx 180 ry 0 rz 90 deg; joints [75.264, -17.389, 83.12, 0, 24.269, 75.264]
  MoveL 1036 to (8.05, 35.8, -1.75) mm, rotated rx 180 ry 0 rz 90 deg; joints [75.05, -17.819, 84.743, 0, 23.076, 75.05]
  MoveL 1037 to (7.11, 35.74, -1.75) mm, rotated rx 180 ry 0 rz 90 deg; joints [75.039, -17.836, 84.809, 0, 23.027, 75.039]
  MoveC 1038 to (3, 34.58, -1.75) mm, rotated rx 180 ry 0 rz 90 deg; joints [74.966, -17.906, 85.079, 0, 22.827, 74.966] to (-0.18, 31.75, -1.75) mm, rotated rx -180 ry 0 rz 90 deg; joints [74.845, -17.95, 85.25, 0, 22.7, 74.845]
  MoveC 1039 to (-1.39, 28.04, -1.75) mm, rotated rx -180 ry 0 rz 90 deg; joints [74.713, -17.953, 85.264, 0, 22.69, 74.713] to (-0.92, 24.17, -1.75) mm, rotated rx 180 ry 0 rz 90 deg; joints [74.591, -17.926, 85.156, 0, 22.77, 74.591]
  MoveL 1040 to (-0.61, 23.22, -1.75) mm, rotated rx -180 ry 0 rz 90 deg; joints [74.563, -17.915, 85.115, 0, 22.8, 74.563]
  MoveL 1041 to (4.89, 8.05, -1.75) mm, rotated rx -180 ry 0 rz 90 deg; joints [74.121, -17.736, 84.424, 0, 23.312, 74.121]
  MoveL 1042 to (5.53, 6.42, -1.75) mm, rotated rx -180 ry 0 rz 90 deg; joints [74.074, -17.715, 84.344, 0, 23.371, 74.074]
  MoveC 1043 to (6.67, 4.39, -1.75) mm, rotated rx -180 ry 0 rz 90 deg; joints [74.019, -17.683, 84.223, 0, 23.46, 74.019] to (8.29, 2.74, -1.75) mm, rotated rx -180 ry 0 rz 90 deg; joints [73.981, -17.644, 84.073, 0, 23.571, 73.981]
  MoveL 1044 to (25.78, -10.86, -1.75) mm, rotated rx 180 ry 0 rz 90 deg; joints [73.708, -17.23, 82.532, 0, 24.698, 73.708]
  MoveC 1045 to (31.78, -12.64, -1.75) mm, rotated rx 180 ry 0 rz 90 deg; joints [73.707, -17.1, 82.059, 0, 25.041, 73.707] to (37.38, -9.86, -1.75) mm, rotated rx 180 ry 0 rz 90 deg; joints [73.847, -17.003, 81.709, 0, 25.294, 73.847]
  MoveL 1046 to (38.16, -9, -1.75) mm, rotated rx 180 ry 0 rz 90 deg; joints [73.881, -16.992, 81.67, 0, 25.322, 73.881]
  MoveL 1047 to (38.38, -8.72, -1.75) mm, rotated rx 180 ry 0 rz 90 deg; joints [73.891, -16.989, 81.66, 0, 25.33, 73.891]
  MoveL 1048 to (60.62, 22.27, -1.75) mm, rotated rx -180 ry 0 rz 90 deg; joints [75.066, -16.706, 80.653, 0, 26.053, 75.066]
  MoveL 1049 to (61.46, 23.48, -1.75) mm, rotated rx 180 ry 0 rz 90 deg; joints [75.111, -16.695, 80.614, 0, 26.081, 75.111]
  MoveC 1050 to (62.75, 25.88, -1.75) mm, rotated rx 180 ry 0 rz 90 deg; joints [75.197, -16.681, 80.565, 0, 26.116, 75.197] to (63.5, 28.51, -1.75) mm, rotated rx -180 ry 0 rz 90 deg; joints [75.286, -16.68, 80.561, 0, 26.119, 75.286]
  MoveC 1051 to (62.7, 33.09, -1.75) mm, rotated rx 180 ry 0 rz 90 deg; joints [75.424, -16.723, 80.71, 0, 26.012, 75.424] to (59.19, 36.14, -1.75) mm, rotated rx 180 ry 0 rz 90 deg; joints [75.492, -16.813, 81.031, 0, 25.783, 75.492]
  MoveC 1052 to (56.88, 36.81, -1.75) mm, rotated rx 180 ry 0 rz 90 deg; joints [75.495, -16.865, 81.215, 0, 25.65, 75.495] to (54.49, 37.03, -1.75) mm, rotated rx 180 ry 0 rz 90 deg; joints [75.482, -16.916, 81.396, 0, 25.52, 75.482]
  MoveL 1053 to (53.54, 37.02, -1.75) mm, rotated rx -180 ry 0 rz 90 deg; joints [75.474, -16.935, 81.466, 0, 25.469, 75.474]
  MoveL 1054 to (30.8, 36.41, -1.75) mm, rotated rx 180 ry 0 rz 90 deg; joints [75.264, -17.389, 83.12, 0, 24.269, 75.264]
  MoveL 1055 to (31, 28.86, -1.75) mm, rotated rx 180 ry 0 rz 90 deg; joints [75.024, -17.346, 82.96, 0, 24.386, 75.024]
  MoveL 1056 to (31, 28.86, 1.25) mm, rotated rx 180 ry 0 rz 90 deg; joints [75.024, -17.499, 83.061, 0, 24.438, 75.024]
  Establecer velocidad (1000.0 mm/s)
  MoveL 1057 to (31, 28.86, 10) mm, rotated rx 180 ry 0 rz 90 deg; joints [75.024, -17.943, 83.352, 0, 24.591, 75.024]
  Establecer velocidad (66.7 mm/s)
  MoveL 1058 to (71.06, -30.55, 10) mm, rotated rx 180 ry 0 rz 90 deg; joints [73.508, -16.745, 79.15, 0, 27.596, 73.508]
  MoveL 1059 to (71.06, -30.55, 1.5) mm, rotated rx 180 ry 0 rz 90 deg; joints [73.508, -16.32, 78.864, 0, 27.456, 73.508]
  MoveL 1060 to (72.57, -30.74, 1.09) mm, rotated rx 180 ry 0 rz 90 deg; joints [73.516, -16.265, 78.733, 0, 27.532, 73.516]
  MoveL 1061 to (74.08, -30.55, 0.69) mm, rotated rx -180 ry 0 rz 90 deg; joints [73.536, -16.212, 78.609, 0, 27.603, 73.536]
  MoveL 1062 to (75.51, -30.04, 0.28) mm, rotated rx -180 ry 0 rz 90 deg; joints [73.564, -16.163, 78.498, 0, 27.665, 73.564]
  MoveL 1063 to (76.79, -29.23, -0.12) mm, rotated rx -180 ry 0 rz 90 deg; joints [73.601, -16.119, 78.405, 0, 27.714, 73.601]
  MoveL 1064 to (77.86, -28.15, -0.53) mm, rotated rx -180 ry 0 rz 90 deg; joints [73.644, -16.082, 78.334, 0, 27.748, 73.644]
  MoveL 1065 to (78.67, -26.86, -0.94) mm, rotated rx 180 ry 0 rz 90 deg; joints [73.691, -16.052, 78.288, 0, 27.764, 73.691]
  MoveL 1066 to (79.16, -25.42, -1.34) mm, rotated rx 180 ry 0 rz 90 deg; joints [73.74, -16.03, 78.268, 0, 27.762, 73.74]
  MoveL 1067 to (79.3, -23.91, -1.75) mm, rotated rx -180 ry 0 rz 90 deg; joints [73.788, -16.016, 78.277, 0, 27.739, 73.788]
  MoveL 1068 to (79.3, -4.7, -1.75) mm, rotated rx 180 ry 0 rz 90 deg; joints [74.381, -16.14, 78.694, 0, 27.446, 74.381]
  MoveC 1069 to (79.09, -1.61, -1.75) mm, rotated rx 180 ry 0 rz 90 deg; joints [74.476, -16.163, 78.775, 0, 27.389, 74.476] to (78.47, 1.42, -1.75) mm, rotated rx -180 ry 0 rz 90 deg; joints [74.564, -16.196, 78.886, 0, 27.31, 74.564]
  MoveC 1070 to (73.44, 6.13, -1.75) mm, rotated rx 180 ry 0 rz 90 deg; joints [74.668, -16.336, 79.364, 0, 26.972, 74.668] to (66.84, 4.17, -1.75) mm, rotated rx 180 ry 0 rz 90 deg; joints [74.55, -16.468, 79.821, 0, 26.647, 74.55]
  MoveC 1071 to (64.89, 2, -1.75) mm, rotated rx 180 ry 0 rz 90 deg; joints [74.465, -16.497, 79.921, 0, 26.576, 74.465] to (63.1, -0.3, -1.75) mm, rotated rx 180 ry 0 rz 90 deg; joints [74.378, -16.522, 80.007, 0, 26.514, 74.378]
  MoveL 1072 to (47.9, -21.19, -1.75) mm, rotated rx 180 ry 0 rz 90 deg; joints [73.587, -16.717, 80.692, 0, 26.025, 73.587]
  MoveC 1073 to (46.32, -26.45, -1.75) mm, rotated rx 180 ry 0 rz 90 deg; joints [73.407, -16.718, 80.693, 0, 26.025, 73.407] to (48.39, -31.53, -1.75) mm, rotated rx 180 ry 0 rz 90 deg; joints [73.268, -16.642, 80.428, 0, 26.214, 73.268]
  MoveL 1074 to (64.5, -49.75, -1.75) mm, rotated rx 180 ry 0 rz 90 deg; joints [72.855, -16.174, 78.811, 0, 27.363, 72.855]
  MoveL 1075 to (65.58, -50.89, -1.75) mm, rotated rx 180 ry 0 rz 90 deg; joints [72.83, -16.143, 78.704, 0, 27.439, 72.83]
  MoveC 1076 to (67.88, -52.76, -1.75) mm, rotated rx 180 ry 0 rz 90 deg; joints [72.794, -16.078, 78.486, 0, 27.592, 72.794] to (70.6, -53.96, -1.75) mm, rotated rx 180 ry 0 rz 90 deg; joints [72.783, -16.009, 78.253, 0, 27.756, 72.783]
  MoveC 1077 to (75.59, -52.92, -1.75) mm, rotated rx -180 ry 0 rz 90 deg; joints [72.862, -15.904, 77.899, 0, 28.005, 72.862] to (78.59, -48.8, -1.75) mm, rotated rx -180 ry 0 rz 90 deg; joints [73.017, -15.864, 77.767, 0, 28.098, 73.017]
  MoveC 1078 to (79.15, -45.99, -1.75) mm, rotated rx -180 ry 0 rz 90 deg; joints [73.108, -15.871, 77.789, 0, 28.082, 73.108] to (79.3, -43.12, -1.75) mm, rotated rx 180 ry 0 rz 90 deg; joints [73.197, -15.887, 77.844, 0, 28.044, 73.197]
  MoveL 1079 to (79.3, -23.91, -1.75) mm, rotated rx -180 ry 0 rz 90 deg; joints [73.788, -16.016, 78.277, 0, 27.739, 73.788]
  MoveL 1080 to (71.75, -23.91, -1.75) mm, rotated rx 180 ry 0 rz 90 deg; joints [73.72, -16.185, 78.85, 0, 27.336, 73.72]
  MoveL 1081 to (71.75, -23.91, 1.25) mm, rotated rx 180 ry 0 rz 90 deg; joints [73.72, -16.336, 78.951, 0, 27.384, 73.72]
  Establecer velocidad (1000.0 mm/s)
  MoveL 1082 to (71.75, -23.91, 10) mm, rotated rx -180 ry 0 rz 90 deg; joints [73.72, -16.774, 79.245, 0, 27.529, 73.72]
  Establecer velocidad (66.7 mm/s)
  MoveL 1083 to (19.03, -72.6, 10) mm, rotated rx 180 ry 0 rz 90 deg; joints [71.696, -17.574, 82.021, 0, 25.553, 71.696]
  MoveL 1084 to (19.03, -72.6, 1.5) mm, rotated rx 180 ry 0 rz 90 deg; joints [71.696, -17.145, 81.738, 0, 25.407, 71.696]
  MoveL 1085 to (18.86, -74.11, 1.09) mm, rotated rx -180 ry 0 rz 90 deg; joints [71.647, -17.118, 81.7, 0, 25.418, 71.647]
  MoveL 1086 to (19.06, -75.61, 0.69) mm, rotated rx -180 ry 0 rz 90 deg; joints [71.602, -17.083, 81.636, 0, 25.447, 71.602]
  MoveL 1087 to (19.59, -77.04, 0.28) mm, rotated rx -180 ry 0 rz 90 deg; joints [71.563, -17.042, 81.55, 0, 25.492, 71.563]
  MoveL 1088 to (20.41, -78.31, -0.12) mm, rotated rx 180 ry 0 rz 90 deg; joints [71.532, -16.996, 81.445, 0, 25.551, 71.532]
  MoveL 1089 to (21.5, -79.37, -0.53) mm, rotated rx 180 ry 0 rz 90 deg; joints [71.51, -16.946, 81.327, 0, 25.62, 71.51]
  MoveL 1090 to (22.8, -80.16, -0.94) mm, rotated rx 180 ry 0 rz 90 deg; joints [71.499, -16.894, 81.2, 0, 25.694, 71.499]
  MoveL 1091 to (24.24, -80.65, -1.34) mm, rotated rx -180 ry 0 rz 90 deg; joints [71.499, -16.841, 81.07, 0, 25.771, 71.499]
  MoveL 1092 to (25.75, -80.77, -1.75) mm, rotated rx 180 ry 0 rz 90 deg; joints [71.511, -16.788, 80.943, 0, 25.846, 71.511]
  MoveL 1093 to (46.91, -80.57, -1.75) mm, rotated rx 180 ry 0 rz 90 deg; joints [71.734, -16.344, 79.391, 0, 26.953, 71.734]
  MoveL 1094 to (53.87, -80.47, -1.75) mm, rotated rx -180 ry 0 rz 90 deg; joints [71.807, -16.193, 78.875, 0, 27.318, 71.807]
  MoveC 1095 to (56.8, -80.05, -1.75) mm, rotated rx -180 ry 0 rz 90 deg; joints [71.85, -16.131, 78.665, 0, 27.466, 71.85] to (59.53, -78.9, -1.75) mm, rotated rx 180 ry 0 rz 90 deg; joints [71.912, -16.079, 78.489, 0, 27.59, 71.912]
  MoveC 1096 to (62.52, -75.28, -1.75) mm, rotated rx -180 ry 0 rz 90 deg; joints [72.053, -16.039, 78.353, 0, 27.686, 72.053] to (62.47, -70.59, -1.75) mm, rotated rx -180 ry 0 rz 90 deg; joints [72.196, -16.074, 78.47, 0, 27.603, 72.196]
  MoveC 1097 to (61.2, -67.94, -1.75) mm, rotated rx 180 ry 0 rz 90 deg; joints [72.264, -16.121, 78.63, 0, 27.491, 72.264] to (59.48, -65.56, -1.75) mm, rotated rx -180 ry 0 rz 90 deg; joints [72.32, -16.176, 78.816, 0, 27.36, 72.32]
  MoveL 1098 to (58.28, -64.16, -1.75) mm, rotated rx 180 ry 0 rz 90 deg; joints [72.352, -16.212, 78.939, 0, 27.272, 72.352]
  MoveL 1099 to (31.89, -33.64, -1.75) mm, rotated rx 180 ry 0 rz 90 deg; joints [73.045, -16.971, 81.594, 0, 25.377, 73.045]
  MoveL 1100 to (30.22, -31.75, -1.75) mm, rotated rx 180 ry 0 rz 90 deg; joints [73.089, -17.017, 81.757, 0, 25.259, 73.089]
  MoveL 1101 to (29.85, -31.39, -1.75) mm, rotated rx -180 ry 0 rz 90 deg; joints [73.096, -17.026, 81.792, 0, 25.234, 73.096]
  MoveL 1102 to (14.69, -19.28, -1.75) mm, rotated rx -180 ry 0 rz 90 deg; joints [73.335, -17.398, 83.153, 0, 24.245, 73.335]
  MoveC 1103 to (11.12, -17.41, -1.75) mm, rotated rx -180 ry 0 rz 90 deg; joints [73.361, -17.478, 83.449, 0, 24.029, 73.361] to (7.11, -17.03, -1.75) mm, rotated rx 180 ry 0 rz 90 deg; joints [73.334, -17.557, 83.744, 0, 23.813, 73.334]
  MoveC 1104 to (2.86, -19.17, -1.75) mm, rotated rx -180 ry 0 rz 90 deg; joints [73.225, -17.625, 84.001, 0, 23.624, 73.225] to (0.36, -23.22, -1.75) mm, rotated rx -180 ry 0 rz 90 deg; joints [73.071, -17.649, 84.091, 0, 23.557, 73.071]
  MoveL 1105 to (0.07, -24.17, -1.75) mm, rotated rx 180 ry 0 rz 90 deg; joints [73.038, -17.649, 84.091, 0, 23.557, 73.038]
  MoveL 1106 to (-12.09, -69.97, -1.75) mm, rotated rx -180 ry 0 rz 90 deg; joints [71.452, -17.602, 83.914, 0, 23.688, 71.452]
  MoveC 1107 to (-11.12, -76.72, -1.75) mm, rotated rx 180 ry 0 rz 90 deg; joints [71.248, -17.541, 83.685, 0, 23.856, 71.248] to (-5.59, -80.71, -1.75) mm, rotated rx 180 ry 0 rz 90 deg; joints [71.182, -17.41, 83.197, 0, 24.213, 71.182]
  MoveC 1108 to (-3.99, -80.97, -1.75) mm, rotated rx -180 ry 0 rz 90 deg; joints [71.191, -17.378, 83.077, 0, 24.301, 71.191] to (-2.37, -81.05, -1.75) mm, rotated rx 180 ry 0 rz 90 deg; joints [71.206, -17.346, 82.961, 0, 24.386, 71.206]
  MoveL 1109 to (25.75, -80.77, -1.75) mm, rotated rx 180 ry 0 rz 90 deg; joints [71.511, -16.788, 80.943, 0, 25.846, 71.511]
  MoveL 1110 to (25.68, -73.22, -1.75) mm, rotated rx 180 ry 0 rz 90 deg; joints [71.745, -16.841, 81.131, 0, 25.711, 71.745]
  MoveL 1111 to (25.68, -73.22, 1.25) mm, rotated rx -180 ry 0 rz 90 deg; joints [71.745, -16.993, 81.232, 0, 25.761, 71.745]
  Establecer velocidad (1000.0 mm/s)
  MoveL 1112 to (25.68, -73.22, 10) mm, rotated rx -180 ry 0 rz 90 deg; joints [71.745, -17.434, 81.524, 0, 25.91, 71.745]
  Establecer velocidad (66.7 mm/s)
  MoveL 1113 to (-60.12, -72.79, 10) mm, rotated rx 180 ry 0 rz 90 deg; joints [70.835, -19.036, 87.558, 0, 21.478, 70.835]
  MoveL 1114 to (-60.12, -72.79, 1.5) mm, rotated rx 180 ry 0 rz 90 deg; joints [70.835, -18.597, 87.276, 0, 21.321, 70.835]
  MoveL 1115 to (-60.29, -74.29, 1.09) mm, rotated rx 180 ry 0 rz 90 deg; joints [70.784, -18.571, 87.239, 0, 21.331, 70.784]
  MoveL 1116 to (-60.1, -75.8, 0.69) mm, rotated rx 180 ry 0 rz 90 deg; joints [70.737, -18.538, 87.177, 0, 21.361, 70.737]
  MoveL 1117 to (-59.57, -77.23, 0.28) mm, rotated rx 180 ry 0 rz 90 deg; joints [70.697, -18.5, 87.094, 0, 21.406, 70.697]
  MoveL 1118 to (-58.75, -78.5, -0.12) mm, rotated rx -180 ry 0 rz 90 deg; joints [70.665, -18.457, 86.994, 0, 21.464, 70.665]
  MoveL 1119 to (-57.66, -79.56, -0.53) mm, rotated rx 180 ry 0 rz 90 deg; joints [70.643, -18.412, 86.881, 0, 21.531, 70.643]
  MoveL 1120 to (-56.36, -80.36, -0.94) mm, rotated rx 180 ry 0 rz 90 deg; joints [70.632, -18.365, 86.76, 0, 21.605, 70.632]
  MoveL 1121 to (-54.92, -80.85, -1.34) mm, rotated rx 180 ry 0 rz 90 deg; joints [70.633, -18.317, 86.637, 0, 21.68, 70.633]
  MoveL 1122 to (-53.41, -80.97, -1.75) mm, rotated rx -180 ry 0 rz 90 deg; joints [70.646, -18.269, 86.517, 0, 21.752, 70.646]
  MoveL 1123 to (-35.28, -80.83, -1.75) mm, rotated rx -180 ry 0 rz 90 deg; joints [70.854, -17.956, 85.275, 0, 22.681, 70.854]
  MoveC 1124 to (-29.03, -78.65, -1.75) mm, rotated rx -180 ry 0 rz 90 deg; joints [70.992, -17.858, 84.893, 0, 22.965, 70.992] to (-25.39, -73.12, -1.75) mm, rotated rx 180 ry 0 rz 90 deg; joints [71.209, -17.827, 84.772, 0, 23.055, 71.209]
  MoveL 1125 to (-12.68, -24.27, -1.75) mm, rotated rx 180 ry 0 rz 90 deg; joints [72.909, -17.883, 84.989, 0, 22.894, 72.909]
  MoveC 1126 to (-12.45, -19.82, -1.75) mm, rotated rx -180 ry 0 rz 90 deg; joints [73.055, -17.903, 85.069, 0, 22.834, 73.055] to (-14.01, -15.64, -1.75) mm, rotated rx 180 ry 0 rz 90 deg; joints [73.175, -17.954, 85.267, 0, 22.687, 73.175]
  MoveC 1127 to (-18.29, -12.29, -1.75) mm, rotated rx -180 ry 0 rz 90 deg; joints [73.242, -18.049, 85.637, 0, 22.411, 73.242] to (-23.69, -11.79, -1.75) mm, rotated rx -180 ry 0 rz 90 deg; joints [73.205, -18.147, 86.025, 0, 22.122, 73.205]
  MoveL 1128 to (-25.11, -12.06, -1.75) mm, rotated rx -180 ry 0 rz 90 deg; joints [73.182, -18.17, 86.118, 0, 22.052, 73.182]
  MoveL 1129 to (-73.68, -22.39, -1.75) mm, rotated rx 180 ry 0 rz 90 deg; joints [72.344, -18.912, 89.211, 0, 19.701, 72.344]
  MoveC 1130 to (-79.48, -25.95, -1.75) mm, rotated rx -180 ry 0 rz 90 deg; joints [72.164, -18.983, 89.523, 0, 19.46, 72.164] to (-81.75, -32.36, -1.75) mm, rotated rx 180 ry 0 rz 90 deg; joints [71.925, -18.986, 89.536, 0, 19.45, 71.925]
  MoveL 1131 to (-81.75, -71, -1.75) mm, rotated rx 180 ry 0 rz 90 deg; joints [70.647, -18.786, 88.664, 0, 20.122, 70.647]
  MoveC 1132 to (-78.75, -78.18, -1.75) mm, rotated rx -180 ry 0 rz 90 deg; joints [70.446, -18.699, 88.295, 0, 20.405, 70.446] to (-71.55, -81.12, -1.75) mm, rotated rx 180 ry 0 rz 90 deg; joints [70.434, -18.568, 87.741, 0, 20.826, 70.434]
  MoveL 1133 to (-53.41, -80.97, -1.75) mm, rotated rx -180 ry 0 rz 90 deg; joints [70.646, -18.269, 86.517, 0, 21.752, 70.646]
  MoveL 1134 to (-53.47, -73.42, -1.75) mm, rotated rx -180 ry 0 rz 90 deg; joints [70.889, -18.315, 86.701, 0, 21.614, 70.889]
  MoveL 1135 to (-53.47, -73.42, 1.25) mm, rotated rx -180 ry 0 rz 90 deg; joints [70.889, -18.47, 86.801, 0, 21.668, 70.889]
  Establecer velocidad (1000.0 mm/s)
  MoveL 1136 to (-53.47, -73.42, 10) mm, rotated rx 180 ry 0 rz 90 deg; joints [70.889, -18.921, 87.092, 0, 21.829, 70.889]
  Establecer velocidad (66.7 mm/s)
  MoveL 1137 to (-73.51, 36.2, 10) mm, rotated rx -180 ry 0 rz 90 deg; joints [74.32, -19.789, 90.765, 0, 19.024, 74.32]
  MoveL 1138 to (-73.51, 36.2, 1.5) mm, rotated rx -180 ry 0 rz 90 deg; joints [74.32, -19.344, 90.483, 0, 18.861, 74.32]
  MoveL 1139 to (-75.01, 36.39, 1.09) mm, rotated rx 180 ry 0 rz 90 deg; joints [74.312, -19.345, 90.573, 0, 18.772, 74.312]
  MoveL 1140 to (-76.52, 36.21, 0.69) mm, rotated rx 180 ry 0 rz 90 deg; joints [74.291, -19.345, 90.657, 0, 18.688, 74.291]
  MoveL 1141 to (-77.95, 35.69, 0.28) mm, rotated rx 180 ry 0 rz 90 deg; joints [74.26, -19.343, 90.729, 0, 18.614, 74.26]
  MoveL 1142 to (-79.24, 34.88, -0.12) mm, rotated rx 180 ry 0 rz 90 deg; joints [74.22, -19.337, 90.785, 0, 18.551, 74.22]
  MoveL 1143 to (-80.3, 33.8, -0.53) mm, rotated rx -180 ry 0 rz 90 deg; joints [74.172, -19.326, 90.822, 0, 18.504, 74.172]
  MoveL 1144 to (-81.11, 32.51, -0.94) mm, rotated rx -180 ry 0 rz 90 deg; joints [74.121, -19.311, 90.838, 0, 18.473, 74.121]
  MoveL 1145 to (-81.61, 31.07, -1.34) mm, rotated rx 180 ry 0 rz 90 deg; joints [74.067, -19.291, 90.83, 0, 18.461, 74.067]
  MoveL 1146 to (-81.75, 29.56, -1.75) mm, rotated rx -180 ry 0 rz 90 deg; joints [74.014, -19.266, 90.797, 0, 18.468, 74.014]
  MoveL 1147 to (-81.75, 1.42, -1.75) mm, rotated rx -180 ry 0 rz 90 deg; joints [73.059, -19.145, 90.245, 0, 18.9, 73.059]
  MoveL 1148 to (-81.75, 0.47, -1.75) mm, rotated rx 180 ry 0 rz 90 deg; joints [73.027, -19.14, 90.225, 0, 18.915, 73.027]
  MoveC 1149 to (-78.44, -7.04, -1.75) mm, rotated rx 180 ry 0 rz 90 deg; joints [72.808, -19.057, 89.851, 0, 19.206, 72.808] to (-70.6, -9.51, -1.75) mm, rotated rx 180 ry 0 rz 90 deg; joints [72.807, -18.927, 89.276, 0, 19.651, 72.807]
  MoveL 1150 to (-69.65, -9.4, -1.75) mm, rotated rx -180 ry 0 rz 90 deg; joints [72.82, -18.913, 89.215, 0, 19.698, 72.82]
  MoveL 1151 to (-68.7, -9.2, -1.75) mm, rotated rx -180 ry 0 rz 90 deg; joints [72.837, -18.899, 89.155, 0, 19.744, 72.837]
  MoveL 1152 to (-19.14, 2.19, -1.75) mm, rotated rx 180 ry 0 rz 90 deg; joints [73.705, -18.14, 85.997, 0, 22.143, 73.705]
  MoveC 1153 to (-12.78, 6.88, -1.75) mm, rotated rx -180 ry 0 rz 90 deg; joints [73.919, -18.051, 85.647, 0, 22.404, 73.919] to (-11.84, 14.72, -1.75) mm, rotated rx 180 ry 0 rz 90 deg; joints [74.183, -18.074, 85.739, 0, 22.336, 74.183]
  MoveL 1154 to (-12.11, 15.64, -1.75) mm, rotated rx 180 ry 0 rz 90 deg; joints [74.211, -18.084, 85.776, 0, 22.308, 74.211]
  MoveL 1155 to (-18.89, 34.57, -1.75) mm, rotated rx -180 ry 0 rz 90 deg; joints [74.771, -18.294, 86.617, 0, 21.677, 74.771]
  MoveC 1156 to (-20.56, 37.56, -1.75) mm, rotated rx -180 ry 0 rz 90 deg; joints [74.855, -18.337, 86.789, 0, 21.547, 74.855] to (-23.1, 39.85, -1.75) mm, rotated rx -180 ry 0 rz 90 deg; joints [74.908, -18.391, 87.009, 0, 21.382, 74.908]
  MoveL 1157 to (-65.86, 67.27, -1.75) mm, rotated rx 180 ry 0 rz 90 deg; joints [75.45, -19.184, 90.424, 0, 18.76, 75.45]
  MoveC 1158 to (-69.06, 68.67, -1.75) mm, rotated rx -180 ry 0 rz 90 deg; joints [75.47, -19.236, 90.663, 0, 18.574, 75.47] to (-72.52, 69.15, -1.75) mm, rotated rx -180 ry 0 rz 90 deg; joints [75.456, -19.288, 90.902, 0, 18.386, 75.456]
  MoveC 1159 to (-77.91, 67.36, -1.75) mm, rotated rx 180 ry 0 rz 90 deg; joints [75.346, -19.359, 91.231, 0, 18.128, 75.346] to (-81.16, 62.7, -1.75) mm, rotated rx 180 ry 0 rz 90 deg; joints [75.156, -19.387, 91.365, 0, 18.022, 75.156]
  MoveC 1160 to (-81.6, 60.7, -1.75) mm, rotated rx 180 ry 0 rz 90 deg; joints [75.083, -19.386, 91.359, 0, 18.027, 75.083] to (-81.75, 58.65, -1.75) mm, rotated rx 180 ry 0 rz 90 deg; joints [75.011, -19.38, 91.332, 0, 18.048, 75.011]
  MoveL 1161 to (-81.75, 29.56, -1.75) mm, rotated rx -180 ry 0 rz 90 deg; joints [74.014, -19.266, 90.797, 0, 18.468, 74.014]
  MoveL 1162 to (-74.2, 29.56, -1.75) mm, rotated rx -180 ry 0 rz 90 deg; joints [74.087, -19.156, 90.294, 0, 18.861, 74.087]
  MoveL 1163 to (-74.2, 29.56, 1.25) mm, rotated rx 180 ry 0 rz 90 deg; joints [74.087, -19.313, 90.395, 0, 18.918, 74.087]
  Establecer velocidad (1000.0 mm/s)
  MoveL 1164 to (-74.2, 29.56, 10) mm, rotated rx 180 ry 0 rz 90 deg; joints [74.087, -19.772, 90.686, 0, 19.086, 74.087]
  Establecer velocidad (66.7 mm/s)
  MoveL 1165 to (-73.01, 36.2, 10) mm, rotated rx -180 ry 0 rz 90 deg; joints [74.325, -19.782, 90.732, 0, 19.05, 74.325]
  MoveL 1166 to (-73.01, 36.2, 1.25) mm, rotated rx -180 ry 0 rz 90 deg; joints [74.325, -19.323, 90.441, 0, 18.882, 74.325]
  MoveL 1167 to (-74.51, 36.39, 0.84) mm, rotated rx -180 ry 0 rz 90 deg; joints [74.316, -19.325, 90.531, 0, 18.793, 74.316]
  MoveL 1168 to (-76.02, 36.21, 0.44) mm, rotated rx -180 ry 0 rz 90 deg; joints [74.296, -19.325, 90.615, 0, 18.71, 74.296]
  MoveL 1169 to (-77.45, 35.69, 0.03) mm, rotated rx -180 ry 0 rz 90 deg; joints [74.265, -19.322, 90.687, 0, 18.635, 74.265]
  MoveL 1170 to (-78.73, 34.88, -0.38) mm, rotated rx 180 ry 0 rz 90 deg; joints [74.224, -19.316, 90.744, 0, 18.572, 74.224]
  MoveL 1171 to (-79.8, 33.8, -0.78) mm, rotated rx 180 ry 0 rz 90 deg; joints [74.177, -19.306, 90.781, 0, 18.525, 74.177]
  MoveL 1172 to (-80.61, 32.51, -1.19) mm, rotated rx -180 ry 0 rz 90 deg; joints [74.126, -19.291, 90.796, 0, 18.494, 74.126]
  MoveL 1173 to (-81.11, 31.07, -1.59) mm, rotated rx -180 ry 0 rz 90 deg; joints [74.072, -19.271, 90.789, 0, 18.482, 74.072]
  MoveL 1174 to (-81.25, 29.56, -2) mm, rotated rx 180 ry 0 rz 90 deg; joints [74.019, -19.245, 90.756, 0, 18.49, 74.019]
  MoveL 1175 to (-81.25, 0.47, -2) mm, rotated rx 180 ry 0 rz 90 deg; joints [73.032, -19.12, 90.184, 0, 18.936, 73.032]
  MoveC 1176 to (-78.09, -6.69, -2) mm, rotated rx -180 ry 0 rz 90 deg; joints [72.824, -19.04, 89.827, 0, 19.214, 72.824] to (-70.6, -8.99, -2) mm, rotated rx -180 ry 0 rz 90 deg; joints [72.824, -18.916, 89.278, 0, 19.638, 72.824]
  MoveL 1177 to (-69.65, -8.88, -2) mm, rotated rx -180 ry 0 rz 90 deg; joints [72.837, -18.902, 89.217, 0, 19.685, 72.837]
  MoveL 1178 to (-63.02, -7.4, -2) mm, rotated rx -180 ry 0 rz 90 deg; joints [72.955, -18.807, 88.802, 0, 20.005, 72.955]
  MoveL 1179 to (-19.43, 2.64, -2) mm, rotated rx 180 ry 0 rz 90 deg; joints [73.717, -18.134, 86.018, 0, 22.116, 73.717]
  MoveC 1180 to (-13.22, 7.1, -2) mm, rotated rx 180 ry 0 rz 90 deg; joints [73.922, -18.047, 85.674, 0, 22.373, 73.922] to (-12.33, 14.69, -2) mm, rotated rx 180 ry 0 rz 90 deg; joints [74.178, -18.07, 85.764, 0, 22.306, 74.178]
  MoveL 1181 to (-12.64, 15.64, -2) mm, rotated rx -180 ry 0 rz 90 deg; joints [74.206, -18.08, 85.805, 0, 22.276, 74.206]
  MoveL 1182 to (-19.08, 33.64, -2) mm, rotated rx -180 ry 0 rz 90 deg; joints [74.739, -18.28, 86.604, 0, 21.676, 74.739]
  MoveL 1183 to (-19.43, 34.59, -2) mm, rotated rx -180 ry 0 rz 90 deg; joints [74.767, -18.291, 86.646, 0, 21.644, 74.767]
  MoveC 1184 to (-20.95, 37.26, -2) mm, rotated rx 180 ry 0 rz 90 deg; joints [74.841, -18.329, 86.803, 0, 21.526, 74.841] to (-23.22, 39.33, -2) mm, rotated rx 180 ry 0 rz 90 deg; joints [74.89, -18.377, 86.999, 0, 21.378, 74.89]
  MoveL 1185 to (-24.17, 39.96, -2) mm, rotated rx 180 ry 0 rz 90 deg; joints [74.902, -18.396, 87.077, 0, 21.32, 74.902]
  MoveL 1186 to (-64.91, 66.11, -2) mm, rotated rx 180 ry 0 rz 90 deg; joints [75.419, -19.153, 90.331, 0, 18.821, 75.419]
  MoveL 1187 to (-65.86, 66.69, -2) mm, rotated rx 180 ry 0 rz 90 deg; joints [75.43, -19.169, 90.405, 0, 18.764, 75.43]
  MoveC 1188 to (-69.04, 68.14, -2) mm, rotated rx -180 ry 0 rz 90 deg; joints [75.452, -19.221, 90.644, 0, 18.577, 75.452] to (-72.49, 68.66, -2) mm, rotated rx -180 ry 0 rz 90 deg; joints [75.439, -19.273, 90.884, 0, 18.389, 75.439]
  MoveC 1189 to (-77.41, 67.1, -2) mm, rotated rx -180 ry 0 rz 90 deg; joints [75.341, -19.337, 91.184, 0, 18.153, 75.341] to (-80.52, 62.99, -2) mm, rotated rx 180 ry 0 rz 90 deg; joints [75.171, -19.366, 91.319, 0, 18.047, 75.171]
  MoveC 1190 to (-81.06, 60.89, -2) mm, rotated rx 180 ry 0 rz 90 deg; joints [75.094, -19.366, 91.318, 0, 18.048, 75.094] to (-81.25, 58.74, -2) mm, rotated rx -180 ry 0 rz 90 deg; joints [75.018, -19.36, 91.292, 0, 18.068, 75.018]
  MoveL 1191 to (-81.25, 29.56, -2) mm, rotated rx 180 ry 0 rz 90 deg; joints [74.019, -19.245, 90.756, 0, 18.49, 74.019]
  MoveL 1192 to (-73.7, 29.56, -2) mm, rotated rx 180 ry 0 rz 90 deg; joints [74.092, -19.135, 90.253, 0, 18.883, 74.092]
  MoveL 1193 to (-73.7, 29.56, 1) mm, rotated rx -180 ry 0 rz 90 deg; joints [74.092, -19.292, 90.353, 0, 18.939, 74.092]
  Establecer velocidad (1000.0 mm/s)
  MoveL 1194 to (-73.7, 29.56, 10) mm, rotated rx -180 ry 0 rz 90 deg; joints [74.092, -19.764, 90.652, 0, 19.112, 74.092]
  Establecer velocidad (66.7 mm/s)
  MoveL 1195 to (-73.01, -45.03, 10) mm, rotated rx -180 ry 0 rz 90 deg; joints [71.6, -19.399, 89.064, 0, 20.335, 71.6]
  MoveL 1196 to (-73.01, -45.03, 1.25) mm, rotated rx 180 ry 0 rz 90 deg; joints [71.6, -18.944, 88.773, 0, 20.171, 71.6]
  MoveL 1197 to (-74.51, -44.85, 0.84) mm, rotated rx -180 ry 0 rz 90 deg; joints [71.59, -18.947, 88.865, 0, 20.082, 71.59]
  MoveL 1198 to (-76.02, -45.03, 0.44) mm, rotated rx 180 ry 0 rz 90 deg; joints [71.567, -18.949, 88.948, 0, 20.001, 71.567]
  MoveL 1199 to (-77.45, -45.54, 0.03) mm, rotated rx -180 ry 0 rz 90 deg; joints [71.535, -18.947, 89.019, 0, 19.928, 71.535]
  MoveL 1200 to (-78.73, -46.36, -0.38) mm, rotated rx 180 ry 0 rz 90 deg; joints [71.493, -18.941, 89.073, 0, 19.869, 71.493]
  MoveL 1201 to (-79.8, -47.44, -0.78) mm, rotated rx 180 ry 0 rz 90 deg; joints [71.446, -18.931, 89.106, 0, 19.825, 71.446]
  MoveL 1202 to (-80.61, -48.73, -1.19) mm, rotated rx 180 ry 0 rz 90 deg; joints [71.394, -18.916, 89.117, 0, 19.798, 71.394]
  MoveL 1203 to (-81.11, -50.16, -1.59) mm, rotated rx 180 ry 0 rz 90 deg; joints [71.341, -18.895, 89.105, 0, 19.79, 71.341]
  MoveL 1204 to (-81.25, -51.67, -2) mm, rotated rx 180 ry 0 rz 90 deg; joints [71.289, -18.868, 89.066, 0, 19.802, 71.289]
  MoveL 1205 to (-81.25, -70.96, -2) mm, rotated rx 180 ry 0 rz 90 deg; joints [70.654, -18.765, 88.623, 0, 20.142, 70.654]
  MoveC 1206 to (-78.42, -77.79, -2) mm, rotated rx -180 ry 0 rz 90 deg; joints [70.463, -18.683, 88.273, 0, 20.41, 70.463] to (-71.59, -80.62, -2) mm, rotated rx 180 ry 0 rz 90 deg; joints [70.449, -18.559, 87.748, 0, 20.811, 70.449]
  MoveL 1207 to (-70.6, -80.63, -2) mm, rotated rx 180 ry 0 rz 90 deg; joints [70.461, -18.543, 87.681, 0, 20.861, 70.461]
  MoveL 1208 to (-36.48, -80.35, -2) mm, rotated rx -180 ry 0 rz 90 deg; joints [70.856, -17.968, 85.361, 0, 22.606, 70.856]
  MoveL 1209 to (-35.21, -80.33, -2) mm, rotated rx 180 ry 0 rz 90 deg; joints [70.871, -17.945, 85.274, 0, 22.672, 70.871]
  MoveC 1210 to (-29.46, -78.36, -2) mm, rotated rx -180 ry 0 rz 90 deg; joints [70.997, -17.855, 84.922, 0, 22.933, 70.997] to (-25.98, -73.37, -2) mm, rotated rx -180 ry 0 rz 90 deg; joints [71.194, -17.823, 84.799, 0, 23.024, 71.194]
  MoveL 1211 to (-25.72, -72.49, -2) mm, rotated rx -180 ry 0 rz 90 deg; joints [71.225, -17.824, 84.801, 0, 23.022, 71.225]
  MoveL 1212 to (-13.16, -24.17, -2) mm, rotated rx 180 ry 0 rz 90 deg; joints [72.907, -17.879, 85.017, 0, 22.863, 72.907]
  MoveC 1213 to (-12.97, -19.75, -2) mm, rotated rx 180 ry 0 rz 90 deg; joints [73.052, -17.9, 85.099, 0, 22.802, 73.052] to (-14.61, -15.64, -2) mm, rotated rx 180 ry 0 rz 90 deg; joints [73.169, -17.952, 85.301, 0, 22.651, 73.169]
  MoveC 1214 to (-18.45, -12.75, -2) mm, rotated rx -180 ry 0 rz 90 deg; joints [73.225, -18.036, 85.631, 0, 22.406, 73.225] to (-23.22, -12.23, -2) mm, rotated rx 180 ry 0 rz 90 deg; joints [73.195, -18.123, 85.974, 0, 22.149, 73.195]
  MoveL 1215 to (-24.17, -12.37, -2) mm, rotated rx 180 ry 0 rz 90 deg; joints [73.181, -18.139, 86.037, 0, 22.102, 73.181]
  MoveL 1216 to (-73.53, -22.86, -2) mm, rotated rx -180 ry 0 rz 90 deg; joints [72.331, -18.895, 89.183, 0, 19.712, 72.331]
  MoveC 1217 to (-79.08, -26.26, -2) mm, rotated rx 180 ry 0 rz 90 deg; joints [72.158, -18.963, 89.481, 0, 19.481, 72.158] to (-81.25, -32.39, -2) mm, rotated rx 180 ry 0 rz 90 deg; joints [71.93, -18.965, 89.493, 0, 19.472, 71.93]
  MoveL 1218 to (-81.25, -51.67, -2) mm, rotated rx 180 ry 0 rz 90 deg; joints [71.289, -18.868, 89.066, 0, 19.802, 71.289]
  MoveL 1219 to (-73.7, -51.67, -2) mm, rotated rx 180 ry 0 rz 90 deg; joints [71.374, -18.751, 88.562, 0, 20.189, 71.374]
  MoveL 1220 to (-73.7, -51.67, 1) mm, rotated rx 180 ry 0 rz 90 deg; joints [71.374, -18.907, 88.662, 0, 20.245, 71.374]
  Establecer velocidad (1000.0 mm/s)
  MoveL 1221 to (-73.7, -51.67, 10) mm, rotated rx 180 ry 0 rz 90 deg; joints [71.374, -19.375, 88.961, 0, 20.414, 71.374]
  Establecer velocidad (66.7 mm/s)
  MoveL 1222 to (18.84, -72.1, 10) mm, rotated rx 180 ry 0 rz 90 deg; joints [71.709, -17.581, 82.047, 0, 25.535, 71.709]
  MoveL 1223 to (18.84, -72.1, 1.25) mm, rotated rx 180 ry 0 rz 90 deg; joints [71.709, -17.139, 81.755, 0, 25.384, 71.709]
  MoveL 1224 to (18.67, -73.61, 0.84) mm, rotated rx -180 ry 0 rz 90 deg; joints [71.66, -17.112, 81.718, 0, 25.395, 71.66]
  MoveL 1225 to (18.87, -75.12, 0.44) mm, rotated rx -180 ry 0 rz 90 deg; joints [71.615, -17.078, 81.653, 0, 25.424, 71.615]
  MoveL 1226 to (19.4, -76.54, 0.03) mm, rotated rx -180 ry 0 rz 90 deg; joints [71.576, -17.037, 81.567, 0, 25.47, 71.576]
  MoveL 1227 to (20.23, -77.82, -0.38) mm, rotated rx 180 ry 0 rz 90 deg; joints [71.545, -16.991, 81.463, 0, 25.528, 71.545]
  MoveL 1228 to (21.32, -78.87, -0.78) mm, rotated rx -180 ry 0 rz 90 deg; joints [71.524, -16.941, 81.344, 0, 25.597, 71.524]
  MoveL 1229 to (22.61, -79.66, -1.19) mm, rotated rx 180 ry 0 rz 90 deg; joints [71.513, -16.889, 81.217, 0, 25.672, 71.513]
  MoveL 1230 to (24.05, -80.15, -1.59) mm, rotated rx -180 ry 0 rz 90 deg; joints [71.512, -16.835, 81.087, 0, 25.749, 71.512]
  MoveL 1231 to (25.57, -80.27, -2) mm, rotated rx -180 ry 0 rz 90 deg; joints [71.524, -16.783, 80.96, 0, 25.823, 71.524]
  MoveL 1232 to (51.65, -80, -2) mm, rotated rx -180 ry 0 rz 90 deg; joints [71.799, -16.232, 79.044, 0, 27.188, 71.799]
  MoveL 1233 to (53.88, -79.96, -2) mm, rotated rx 180 ry 0 rz 90 deg; joints [71.823, -16.184, 78.878, 0, 27.305, 71.823]
  MoveC 1234 to (56.31, -79.66, -2) mm, rotated rx 180 ry 0 rz 90 deg; joints [71.857, -16.133, 78.704, 0, 27.429, 71.857] to (58.62, -78.84, -2) mm, rotated rx -180 ry 0 rz 90 deg; joints [71.905, -16.087, 78.551, 0, 27.537, 71.905]
  MoveC 1235 to (61.91, -75.28, -2) mm, rotated rx -180 ry 0 rz 90 deg; joints [72.047, -16.04, 78.39, 0, 27.65, 72.047] to (61.88, -70.43, -2) mm, rotated rx 180 ry 0 rz 90 deg; joints [72.195, -16.076, 78.511, 0, 27.565, 72.195]
  MoveC 1236 to (60.74, -68.15, -2) mm, rotated rx -180 ry 0 rz 90 deg; joints [72.253, -16.117, 78.651, 0, 27.466, 72.253] to (59.25, -66.09, -2) mm, rotated rx 180 ry 0 rz 90 deg; joints [72.302, -16.165, 78.813, 0, 27.352, 72.302]
  MoveL 1237 to (56.62, -63.02, -2) mm, rotated rx 180 ry 0 rz 90 deg; joints [72.371, -16.244, 79.083, 0, 27.161, 72.371]
  MoveL 1238 to (32.07, -34.59, -2) mm, rotated rx -180 ry 0 rz 90 deg; joints [73.017, -16.949, 81.551, 0, 25.398, 73.017]
  MoveL 1239 to (29.85, -32.08, -2) mm, rotated rx 180 ry 0 rz 90 deg; joints [73.075, -17.009, 81.769, 0, 25.241, 73.075]
  MoveL 1240 to (29.5, -31.75, -2) mm, rotated rx -180 ry 0 rz 90 deg; joints [73.082, -17.018, 81.801, 0, 25.217, 73.082]
  MoveL 1241 to (14.69, -19.89, -2) mm, rotated rx 180 ry 0 rz 90 deg; joints [73.316, -17.382, 83.131, 0, 24.251, 73.316]
  MoveL 1242 to (13.63, -19.15, -2) mm, rotated rx -180 ry 0 rz 90 deg; joints [73.329, -17.407, 83.223, 0, 24.184, 73.329]
  MoveC 1243 to (10.05, -17.65, -2) mm, rotated rx -180 ry 0 rz 90 deg; joints [73.343, -17.484, 83.512, 0, 23.972, 73.343] to (6.16, -17.76, -2) mm, rotated rx 180 ry 0 rz 90 deg; joints [73.302, -17.558, 83.787, 0, 23.77, 73.302]
  MoveC 1244 to (2.87, -19.87, -2) mm, rotated rx 180 ry 0 rz 90 deg; joints [73.203, -17.608, 83.977, 0, 23.631, 73.203] to (0.88, -23.22, -2) mm, rotated rx -180 ry 0 rz 90 deg; joints [73.076, -17.626, 84.046, 0, 23.58, 73.076]
  MoveL 1245 to (0.58, -24.17, -2) mm, rotated rx 180 ry 0 rz 90 deg; joints [73.043, -17.626, 84.046, 0, 23.58, 73.043]
  MoveL 1246 to (-11.5, -69.65, -2) mm, rotated rx 180 ry 0 rz 90 deg; joints [71.468, -17.58, 83.871, 0, 23.709, 71.468]
  MoveL 1247 to (-11.69, -70.6, -2) mm, rotated rx 180 ry 0 rz 90 deg; joints [71.436, -17.578, 83.863, 0, 23.715, 71.436]
  MoveC 1248 to (-10.99, -75.93, -2) mm, rotated rx -180 ry 0 rz 90 deg; joints [71.275, -17.531, 83.686, 0, 23.845, 71.275] to (-7.11, -79.65, -2) mm, rotated rx 180 ry 0 rz 90 deg; joints [71.199, -17.433, 83.322, 0, 24.111, 71.199]
  MoveC 1249 to (-4.98, -80.35, -2) mm, rotated rx -180 ry 0 rz 90 deg; joints [71.2, -17.388, 83.154, 0, 24.234, 71.2] to (-2.75, -80.57, -2) mm, rotated rx 180 ry 0 rz 90 deg; joints [71.217, -17.344, 82.991, 0, 24.354, 71.217]
  MoveL 1250 to (25.57, -80.27, -2) mm, rotated rx -180 ry 0 rz 90 deg; joints [71.524, -16.783, 80.96, 0, 25.823, 71.524]
  MoveL 1251 to (25.49, -72.72, -2) mm, rotated rx -180 ry 0 rz 90 deg; joints [71.758, -16.836, 81.148, 0, 25.688, 71.758]
  MoveL 1252 to (25.49, -72.72, 1) mm, rotated rx 180 ry 0 rz 90 deg; joints [71.758, -16.987, 81.249, 0, 25.738, 71.758]
  Establecer velocidad (1000.0 mm/s)
  MoveL 1253 to (25.49, -72.72, 10) mm, rotated rx 180 ry 0 rz 90 deg; joints [71.758, -17.441, 81.55, 0, 25.891, 71.758]
  Establecer velocidad (66.7 mm/s)
  MoveL 1254 to (70.57, -30.77, 10) mm, rotated rx 180 ry 0 rz 90 deg; joints [73.497, -16.755, 79.182, 0, 27.573, 73.497]
  MoveL 1255 to (70.57, -30.77, 1.25) mm, rotated rx 180 ry 0 rz 90 deg; joints [73.497, -16.317, 78.888, 0, 27.429, 73.497]
  MoveL 1256 to (72.08, -30.95, 0.84) mm, rotated rx 180 ry 0 rz 90 deg; joints [73.505, -16.262, 78.757, 0, 27.505, 73.505]
  MoveL 1257 to (73.59, -30.77, 0.44) mm, rotated rx 180 ry 0 rz 90 deg; joints [73.524, -16.209, 78.633, 0, 27.576, 73.524]
  MoveL 1258 to (75.02, -30.26, 0.03) mm, rotated rx -180 ry 0 rz 90 deg; joints [73.553, -16.16, 78.522, 0, 27.638, 73.553]
  MoveL 1259 to (76.3, -29.44, -0.38) mm, rotated rx 180 ry 0 rz 90 deg; joints [73.59, -16.116, 78.429, 0, 27.687, 73.59]
  MoveL 1260 to (77.37, -28.36, -0.78) mm, rotated rx 180 ry 0 rz 90 deg; joints [73.633, -16.079, 78.358, 0, 27.721, 73.633]
  MoveL 1261 to (78.17, -27.07, -1.19) mm, rotated rx 180 ry 0 rz 90 deg; joints [73.68, -16.049, 78.312, 0, 27.737, 73.68]
  MoveL 1262 to (78.67, -25.64, -1.59) mm, rotated rx 180 ry 0 rz 90 deg; joints [73.729, -16.027, 78.292, 0, 27.735, 73.729]
  MoveL 1263 to (78.81, -24.13, -2) mm, rotated rx 180 ry 0 rz 90 deg; joints [73.777, -16.014, 78.301, 0, 27.712, 73.777]
  MoveL 1264 to (78.81, -4.61, -2) mm, rotated rx -180 ry 0 rz 90 deg; joints [74.38, -16.139, 78.724, 0, 27.414, 74.38]
  MoveC 1265 to (78.68, -2.2, -2) mm, rotated rx -180 ry 0 rz 90 deg; joints [74.454, -16.157, 78.786, 0, 27.371, 74.454] to (78.28, 0.17, -2) mm, rotated rx -180 ry 0 rz 90 deg; joints [74.524, -16.18, 78.866, 0, 27.314, 74.524]
  MoveC 1266 to (74.85, 4.73, -2) mm, rotated rx 180 ry 0 rz 90 deg; joints [74.636, -16.284, 79.221, 0, 27.063, 74.636] to (69.16, 5.21, -2) mm, rotated rx -180 ry 0 rz 90 deg; joints [74.603, -16.411, 79.659, 0, 26.752, 74.603]
  MoveC 1267 to (66.84, 3.49, -2) mm, rotated rx -180 ry 0 rz 90 deg; joints [74.529, -16.452, 79.798, 0, 26.653, 74.529] to (64.91, 1.32, -2) mm, rotated rx -180 ry 0 rz 90 deg; joints [74.444, -16.48, 79.897, 0, 26.583, 74.444]
  MoveL 1268 to (48.38, -21.32, -2) mm, rotated rx 180 ry 0 rz 90 deg; joints [73.587, -16.694, 80.645, 0, 26.049, 73.587]
  MoveC 1269 to (46.82, -26.36, -2) mm, rotated rx 180 ry 0 rz 90 deg; joints [73.415, -16.695, 80.65, 0, 26.045, 73.415] to (48.8, -31.24, -2) mm, rotated rx -180 ry 0 rz 90 deg; joints [73.281, -16.623, 80.395, 0, 26.228, 73.281]
  MoveL 1270 to (50.7, -33.39, -2) mm, rotated rx -180 ry 0 rz 90 deg; joints [73.231, -16.569, 80.207, 0, 26.362, 73.231]
  MoveL 1271 to (64.91, -49.46, -2) mm, rotated rx 180 ry 0 rz 90 deg; joints [72.868, -16.155, 78.779, 0, 27.376, 72.868]
  MoveL 1272 to (65.67, -50.27, -2) mm, rotated rx 180 ry 0 rz 90 deg; joints [72.85, -16.132, 78.703, 0, 27.429, 72.85]
  MoveC 1273 to (67.52, -51.9, -2) mm, rotated rx -180 ry 0 rz 90 deg; joints [72.817, -16.08, 78.526, 0, 27.554, 72.817] to (69.65, -53.12, -2) mm, rotated rx -180 ry 0 rz 90 deg; joints [72.8, -16.024, 78.336, 0, 27.688, 72.8]
  MoveC 1274 to (74.92, -52.55, -2) mm, rotated rx 180 ry 0 rz 90 deg; joints [72.868, -15.909, 77.95, 0, 27.959, 72.868] to (78.19, -48.37, -2) mm, rotated rx 180 ry 0 rz 90 deg; joints [73.026, -15.864, 77.799, 0, 28.065, 73.026]
  MoveC 1275 to (78.66, -46.03, -2) mm, rotated rx 180 ry 0 rz 90 deg; joints [73.102, -15.87, 77.818, 0, 28.052, 73.102] to (78.81, -43.64, -2) mm, rotated rx -180 ry 0 rz 90 deg; joints [73.177, -15.883, 77.861, 0, 28.022, 73.177]
  MoveL 1276 to (78.81, -24.13, -2) mm, rotated rx 180 ry 0 rz 90 deg; joints [73.777, -16.014, 78.301, 0, 27.712, 73.777]
  MoveL 1277 to (71.26, -24.13, -2) mm, rotated rx -180 ry 0 rz 90 deg; joints [73.709, -16.182, 78.873, 0, 27.309, 73.709]
  MoveL 1278 to (71.26, -24.13, 1) mm, rotated rx 180 ry 0 rz 90 deg; joints [73.709, -16.333, 78.975, 0, 27.358, 73.709]
  Establecer velocidad (1000.0 mm/s)
  MoveL 1279 to (71.26, -24.13, 10) mm, rotated rx -180 ry 0 rz 90 deg; joints [73.709, -16.783, 79.277, 0, 27.506, 73.709]
  Establecer velocidad (66.7 mm/s)
  MoveL 1280 to (38.57, 6.53, 10) mm, rotated rx 180 ry 0 rz 90 deg; joints [74.377, -17.668, 82.356, 0, 25.312, 74.377]
  MoveL 1281 to (38.57, 6.53, 1.25) mm, rotated rx -180 ry 0 rz 90 deg; joints [74.377, -17.225, 82.064, 0, 25.161, 74.377]
  MoveL 1282 to (39.68, 5.5, 0.84) mm, rotated rx 180 ry 0 rz 90 deg; joints [74.354, -17.176, 81.948, 0, 25.228, 74.354]
  MoveL 1283 to (41.02, 4.77, 0.44) mm, rotated rx 180 ry 0 rz 90 deg; joints [74.343, -17.124, 81.822, 0, 25.303, 74.343]
  MoveL 1284 to (42.48, 4.35, 0.03) mm, rotated rx 180 ry 0 rz 90 deg; joints [74.342, -17.072, 81.692, 0, 25.38, 74.342]
  MoveL 1285 to (44, 4.27, -0.38) mm, rotated rx 180 ry 0 rz 90 deg; joints [74.353, -17.02, 81.565, 0, 25.454, 74.353]
  MoveL 1286 to (45.49, 4.52, -0.78) mm, rotated rx 180 ry 0 rz 90 deg; joints [74.374, -16.97, 81.447, 0, 25.523, 74.374]
  MoveL 1287 to (46.9, 5.1, -1.19) mm, rotated rx 180 ry 0 rz 90 deg; joints [74.405, -16.923, 81.341, 0, 25.582, 74.405]
  MoveL 1288 to (48.14, 5.98, -1.59) mm, rotated rx 180 ry 0 rz 90 deg; joints [74.444, -16.882, 81.254, 0, 25.628, 74.444]
  MoveL 1289 to (49.14, 7.12, -2) mm, rotated rx 180 ry 0 rz 90 deg; joints [74.489, -16.848, 81.19, 0, 25.658, 74.489]
  MoveL 1290 to (60.87, 23.48, -2) mm, rotated rx -180 ry 0 rz 90 deg; joints [75.106, -16.695, 80.65, 0, 26.046, 75.106]
  MoveC 1291 to (62.19, 25.84, -2) mm, rotated rx 180 ry 0 rz 90 deg; joints [75.191, -16.68, 80.598, 0, 26.083, 75.191] to (62.96, 28.42, -2) mm, rotated rx -180 ry 0 rz 90 deg; joints [75.279, -16.679, 80.591, 0, 26.088, 75.279]
  MoveC 1292 to (62.28, 32.71, -2) mm, rotated rx -180 ry 0 rz 90 deg; joints [75.409, -16.717, 80.725, 0, 25.991, 75.409] to (59.07, 35.63, -2) mm, rotated rx 180 ry 0 rz 90 deg; joints [75.475, -16.8, 81.021, 0, 25.779, 75.475]
  MoveC 1293 to (56.83, 36.31, -2) mm, rotated rx -180 ry 0 rz 90 deg; joints [75.478, -16.851, 81.201, 0, 25.65, 75.478] to (54.49, 36.52, -2) mm, rotated rx -180 ry 0 rz 90 deg; joints [75.466, -16.9, 81.378, 0, 25.523, 75.466]
  MoveL 1294 to (47.86, 36.36, -2) mm, rotated rx 180 ry 0 rz 90 deg; joints [75.406, -17.036, 81.864, 0, 25.172, 75.406]
  MoveL 1295 to (7.62, 35.29, -2) mm, rotated rx 180 ry 0 rz 90 deg; joints [75.029, -17.812, 84.756, 0, 23.056, 75.029]
  MoveC 1296 to (4.62, 34.74, -2) mm, rotated rx 180 ry 0 rz 90 deg; joints [74.985, -17.864, 84.958, 0, 22.906, 74.985] to (1.94, 33.29, -2) mm, rotated rx -180 ry 0 rz 90 deg; joints [74.914, -17.906, 85.121, 0, 22.785, 74.914]
  MoveC 1297 to (-0.57, 29.84, -2) mm, rotated rx 180 ry 0 rz 90 deg; joints [74.779, -17.935, 85.232, 0, 22.702, 74.779] to (-0.75, 25.58, -2) mm, rotated rx -180 ry 0 rz 90 deg; joints [74.639, -17.917, 85.163, 0, 22.754, 74.639]
  MoveL 1298 to (-0.39, 24.17, -2) mm, rotated rx -180 ry 0 rz 90 deg; joints [74.596, -17.903, 85.11, 0, 22.793, 74.596]
  MoveL 1299 to (5.81, 7.02, -2) mm, rotated rx 180 ry 0 rz 90 deg; joints [74.096, -17.7, 84.329, 0, 23.372, 74.096]
  MoveC 1300 to (6.97, 4.84, -2) mm, rotated rx 180 ry 0 rz 90 deg; joints [74.036, -17.667, 84.202, 0, 23.466, 74.036] to (8.69, 3.06, -2) mm, rotated rx 180 ry 0 rz 90 deg; joints [73.995, -17.625, 84.042, 0, 23.583, 73.995]
  MoveL 1301 to (26.09, -10.46, -2) mm, rotated rx -180 ry 0 rz 90 deg; joints [73.723, -17.214, 82.51, 0, 24.704, 73.723]
  MoveC 1302 to (31.97, -12.11, -2) mm, rotated rx 180 ry 0 rz 90 deg; joints [73.725, -17.087, 82.048, 0, 25.039, 73.725] to (37.33, -9.18, -2) mm, rotated rx 180 ry 0 rz 90 deg; joints [73.867, -16.995, 81.718, 0, 25.277, 73.867]
  MoveL 1303 to (38.25, -8.05, -2) mm, rotated rx 180 ry 0 rz 90 deg; joints [73.912, -16.983, 81.675, 0, 25.308, 73.912]
  MoveL 1304 to (49.14, 7.12, -2) mm, rotated rx 180 ry 0 rz 90 deg; joints [74.489, -16.848, 81.19, 0, 25.658, 74.489]
  MoveL 1305 to (43, 11.52, -2) mm, rotated rx 180 ry 0 rz 90 deg; joints [74.574, -16.999, 81.732, 0, 25.267, 74.574]
  MoveL 1306 to (43, 11.52, 1) mm, rotated rx 180 ry 0 rz 90 deg; joints [74.574, -17.151, 81.833, 0, 25.318, 74.574]
  Establecer velocidad (1000.0 mm/s)
  MoveL 1307 to (43, 11.52, 10) mm, rotated rx 180 ry 0 rz 90 deg; joints [74.574, -17.606, 82.133, 0, 25.473, 74.574]
  Establecer velocidad (66.7 mm/s)
  MoveL 1308 to (26.9, 71.83, 10) mm, rotated rx 180 ry 0 rz 90 deg; joints [76.379, -18.237, 84.441, 0, 23.796, 76.379]
  MoveL 1309 to (26.9, 71.83, 1.25) mm, rotated rx 180 ry 0 rz 90 deg; joints [76.379, -17.791, 84.15, 0, 23.64, 76.379]
  MoveL 1310 to (27.11, 73.33, 0.84) mm, rotated rx 180 ry 0 rz 90 deg; joints [76.43, -17.773, 84.148, 0, 23.625, 76.43]
  MoveL 1311 to (26.94, 74.84, 0.44) mm, rotated rx 180 ry 0 rz 90 deg; joints [76.478, -17.762, 84.172, 0, 23.59, 76.478]
  MoveL 1312 to (26.45, 76.28, 0.03) mm, rotated rx -180 ry 0 rz 90 deg; joints [76.521, -17.757, 84.219, 0, 23.538, 76.521]
  MoveL 1313 to (25.66, 77.57, -0.38) mm, rotated rx -180 ry 0 rz 90 deg; joints [76.557, -17.758, 84.285, 0, 23.473, 76.557]
  MoveL 1314 to (24.59, 78.66, -0.78) mm, rotated rx 180 ry 0 rz 90 deg; joints [76.584, -17.762, 84.367, 0, 23.395, 76.584]
  MoveL 1315 to (23.31, 79.48, -1.19) mm, rotated rx 180 ry 0 rz 90 deg; joints [76.601, -17.769, 84.459, 0, 23.31, 76.601]
  MoveL 1316 to (21.88, 80, -1.59) mm, rotated rx 180 ry 0 rz 90 deg; joints [76.607, -17.777, 84.557, 0, 23.22, 76.607]
  MoveL 1317 to (20.38, 80.16, -2) mm, rotated rx 180 ry 0 rz 90 deg; joints [76.6, -17.785, 84.654, 0, 23.131, 76.6]
  MoveC 1318 to (-5.21, 80.47, -2) mm, rotated rx 180 ry 0 rz 90 deg; joints [76.408, -18.249, 86.476, 0, 21.772, 76.408] to (-30.8, 80.67, -2) mm, rotated rx -180 ry 0 rz 90 deg; joints [76.206, -18.68, 88.26, 0, 20.42, 76.206]
  MoveC 1319 to (-34.64, 80.35, -2) mm, rotated rx -180 ry 0 rz 90 deg; joints [76.163, -18.741, 88.52, 0, 20.222, 76.163] to (-38.38, 79.4, -2) mm, rotated rx -180 ry 0 rz 90 deg; joints [76.1, -18.797, 88.76, 0, 20.037, 76.1]
